(* PLC project flask_motion_app, Dassault Systèmes ControlBuild 2021x HF2 *)
(* stored: creationDateTime 2023-10-03T16:51:02-01:00 *)

CONFIGURATION flask_motion_app
  VAR_GLOBAL
    weight AT 523 : INT := 150;
    masterPosition AT 17 : REAL := 0.0;
    plc/presConvUp AT 6 : BOOL := false;
    plc/presConvDw AT 7 : BOOL := false;
    plc/masterPosition AT 17 : REAL := 0.0;
    plc/idRead AT 525 : INT := 0;
    plc/mesuredWeight AT 526 : INT := 0;
    plc/bpStart AT 8 : BOOL := false;
    plc/bpAuto AT 9 : BOOL := false;
    plc/bpManu AT 10 : BOOL := false;
    plc/bpEmergencyStop AT 11 : BOOL := false;
    plc/bpStop AT 12 : BOOL := false;
    plc/HomeCmd AT 13 : BOOL := false;
    plc/MoveVelCmd AT 14 : BOOL := false;
    plc/MoveAbsCmd AT 15 : BOOL := false;
    plc/MoveVel1ManualCmd AT 16 : BOOL := false;
    plc/MoveVel2ManualCmd AT 17 : BOOL := false;
    plc/MoveAbs1ManualCmd AT 18 : BOOL := false;
    plc/MoveAbs2ManualCmd AT 19 : BOOL := false;
    plc/StopCmd AT 20 : BOOL := false;
    plc/MovePosition AT 32 : REAL := 0.0;
    plc/MoveSpeed AT 33 : REAL := 100.0;
    plc/MoveAcceleration AT 34 : REAL := 100.0;
    plc/MoveDeceleration AT 35 : REAL := 100.0;
    plc/offsetAxToMa AT 36 : REAL := 0.0;
    plc/gripSyringes AT 21 : BOOL := false;
    plc/Auto AT 22 : BOOL := false;
    plc/Manu AT 23 : BOOL := false;
    plc/run AT 24 : BOOL := false;
    plc/forwardUp AT 25 : BOOL := false;
    plc/backwardUp AT 26 : BOOL := false;
    plc/forwardDw AT 27 : BOOL := false;
    plc/backwardDw AT 28 : BOOL := false;
    plc/ejectBadProd AT 29 : BOOL := false;
    plc/modemanagement/bpStart AT 8 : BOOL := false;
    plc/modemanagement/bpAuto AT 9 : BOOL := false;
    plc/modemanagement/bpManu AT 10 : BOOL := false;
    plc/modemanagement/bpEmergencyStop AT 11 : BOOL := false;
    plc/modemanagement/bpStop AT 12 : BOOL := false;
    plc/modemanagement/Auto AT 22 : BOOL := false;
    plc/modemanagement/Manu AT 23 : BOOL := false;
    plc/modemanagement/run AT 24 : BOOL := false;
    plc/motors/Auto AT 22 : BOOL := false;
    plc/motors/Manu AT 23 : BOOL := false;
    plc/motors/run AT 24 : BOOL := false;
    plc/motors/presConvUp AT 6 : BOOL := false;
    plc/motors/presConvDw AT 7 : BOOL := false;
    plc/motors/masterPosition AT 17 : REAL := 0.0;
    plc/motors/mesuredWeight AT 526 : INT := 0;
    plc/motors/phaseCode AT 527 : INT := 0;
    plc/motors/forwardUp AT 25 : BOOL := false;
    plc/motors/backwardUp AT 26 : BOOL := false;
    plc/motors/forwardDw AT 27 : BOOL := false;
    plc/motors/backwardDw AT 28 : BOOL := false;
    plc/motors/ejectBadProd AT 29 : BOOL := false;
    plc/motors/weihtOk AT 30 : BOOL := false;
    plc/motors/upperLimitOk AT 32 : BOOL := false;
    plc/motors/lowerLimitOk AT 33 : BOOL := false;
    plc/motors/prtSensorConvDw AT 529 : TIME := T#0h0m0s500ms;
    plc/motors/prtSensorConvUp AT 533 : TIME := T#0h0m1s500ms;
    plc/motors/upperLimitWeight AT 537 : INT := 125;
    plc/motors/lowerLimitWeight AT 538 : INT := 115;
    plc/robotctrl/forwardUp AT 25 : BOOL := false;
    plc/robotctrl/backwardUp AT 26 : BOOL := false;
    plc/robotctrl/forwardDw AT 27 : BOOL := false;
    plc/robotctrl/backwardDw AT 28 : BOOL := false;
    plc/robotctrl/presConvUp AT 6 : BOOL := false;
    plc/robotctrl/presConvDw AT 7 : BOOL := false;
    plc/robotctrl/masterPosition AT 17 : REAL := 0.0;
    plc/robotctrl/Auto AT 22 : BOOL := false;
    plc/robotctrl/Manu AT 23 : BOOL := false;
    plc/robotctrl/run AT 24 : BOOL := false;
    plc/robotctrl/weightOk AT 30 : BOOL := false;
    plc/robotctrl/phaseCode AT 527 : INT := 0;
    plc/robotctrl/HomeCmd AT 13 : BOOL := false;
    plc/robotctrl/MoveVelCmd AT 14 : BOOL := false;
    plc/robotctrl/MoveAbsCmd AT 15 : BOOL := false;
    plc/robotctrl/MoveVel1ManualCmd AT 16 : BOOL := false;
    plc/robotctrl/MoveVel2ManualCmd AT 17 : BOOL := false;
    plc/robotctrl/MoveAbs1ManualCmd AT 18 : BOOL := false;
    plc/robotctrl/MoveAbs2ManualCmd AT 19 : BOOL := false;
    plc/robotctrl/StopCmd AT 20 : BOOL := false;
    plc/robotctrl/MovePosition AT 32 : REAL := 0.0;
    plc/robotctrl/MoveSpeed AT 33 : REAL := 100.0;
    plc/robotctrl/MoveAcceleration AT 34 : REAL := 100.0;
    plc/robotctrl/MoveDeceleration AT 35 : REAL := 100.0;
    plc/robotctrl/offsetAxToMa AT 36 : REAL := 0.0;
    plc/robotctrl/gripSyringes AT 21 : BOOL := false;
    plc/robotctrl/endPhase1 AT 37 : REAL := 50.0;
    plc/robotctrl/endPhase2 AT 38 : REAL := 60.0;
    plc/robotctrl/endPhase3 AT 39 : REAL := 150.0;
    plc/robotctrl/endPhase4 AT 40 : REAL := 200.0;
    plc/robotctrl/speedPhase1 AT 41 : REAL := 80.0;
    plc/robotctrl/speedPhase2 AT 42 : REAL := 85.0;
    plc/robotctrl/speedPhase3 AT 43 : REAL := 100.0;
    plc/robotctrl/speedPhase4 AT 44 : REAL := 100.0;
    plc/robotctrl/globalSpeedFactor AT 45 : REAL := 100.0;
    robot6axis_ctrled1/armOrigin AT 27 : ARRAY[1..3] OF REAL := [800.0, 400.0, 0.0];
    robot6axis_ctrled1/profileNr AT 524 : DINT := 0;
    robot6axis_ctrled1/HomeCmd AT 13 : BOOL := false;
    robot6axis_ctrled1/MoveVelCmd AT 14 : BOOL := false;
    robot6axis_ctrled1/MoveAbsCmd AT 15 : BOOL := false;
    robot6axis_ctrled1/MoveVel1ManualCmd AT 16 : BOOL := false;
    robot6axis_ctrled1/MoveVel2ManualCmd AT 17 : BOOL := false;
    robot6axis_ctrled1/MoveAbs1ManualCmd AT 18 : BOOL := false;
    robot6axis_ctrled1/MoveAbs2ManualCmd AT 19 : BOOL := false;
    robot6axis_ctrled1/StopCmd AT 20 : BOOL := false;
    robot6axis_ctrled1/MovePosition AT 32 : REAL := 0.0;
    robot6axis_ctrled1/MoveSpeed AT 33 : REAL := 100.0;
    robot6axis_ctrled1/MoveAcceleration AT 34 : REAL := 100.0;
    robot6axis_ctrled1/MoveDeceleration AT 35 : REAL := 100.0;
    robot6axis_ctrled1/offsetAxToMa AT 36 : REAL := 0.0;
    robot6axis_ctrled1/gripSyringes AT 21 : BOOL := false;
    robot6axis_ctrled1/Auto AT 22 : BOOL := false;
    robot6axis_ctrled1/Manu AT 23 : BOOL := false;
    robot6axis_ctrled1/run AT 24 : BOOL := false;
    robot6axis_ctrled1/armExtrem AT 22 : ARRAY[1..3] OF REAL := [3(0.0)];
    robot6axis_ctrled1/velX AT 21 : REAL := 0.0;
    robot6axis_ctrled1/velY AT 20 : REAL := 0.0;
    robot6axis_ctrled1/velZ AT 19 : REAL := 0.0;
    robot6axis_ctrled1/armInStop AT 5 : BOOL := false;
    robot6axis_ctrled1/masterPosition AT 17 : REAL := 0.0;
    robot6axis_ctrled1/ActualPositionAx AT 18 : REAL := 0.0;
    robot6axis_ctrled1/robot6axis_cams/profileNr AT 524 : DINT := 0;
    robot6axis_ctrled1/robot6axis_cams/HomeCmd AT 13 : BOOL := false;
    robot6axis_ctrled1/robot6axis_cams/MoveVelCmd AT 14 : BOOL := false;
    robot6axis_ctrled1/robot6axis_cams/MoveAbsCmd AT 15 : BOOL := false;
    robot6axis_ctrled1/robot6axis_cams/MoveVel1ManualCmd AT 16 : BOOL := false;
    robot6axis_ctrled1/robot6axis_cams/MoveVel2ManualCmd AT 17 : BOOL := false;
    robot6axis_ctrled1/robot6axis_cams/MoveAbs1ManualCmd AT 18 : BOOL := false;
    robot6axis_ctrled1/robot6axis_cams/MoveAbs2ManualCmd AT 19 : BOOL := false;
    robot6axis_ctrled1/robot6axis_cams/StopCmd AT 20 : BOOL := false;
    robot6axis_ctrled1/robot6axis_cams/MovePosition AT 32 : REAL := 0.0;
    robot6axis_ctrled1/robot6axis_cams/MoveSpeed AT 33 : REAL := 100.0;
    robot6axis_ctrled1/robot6axis_cams/MoveAcceleration AT 34 : REAL := 100.0;
    robot6axis_ctrled1/robot6axis_cams/MoveDeceleration AT 35 : REAL := 100.0;
    robot6axis_ctrled1/robot6axis_cams/offsetAxToMa AT 36 : REAL := 0.0;
    robot6axis_ctrled1/robot6axis_cams/name1 AT 636 : STRING(50) := 'CamAxis1_exa.txt';
    robot6axis_ctrled1/robot6axis_cams/name2 AT 583 : STRING(50) := 'CamAxis2_exa.txt';
    robot6axis_ctrled1/robot6axis_cams/name3 AT 530 : STRING(50) := 'CamAxis3_exa.txt';
    robot6axis_ctrled1/robot6axis_cams/name4 AT 477 : STRING(50) := 'CamAxis4_exa.txt';
    robot6axis_ctrled1/robot6axis_cams/name5 AT 424 : STRING(50) := 'CamAxis5_exa.txt';
    robot6axis_ctrled1/robot6axis_cams/name6 AT 371 : STRING(50) := 'CamAxis6_exa.txt';
    robot6axis_ctrled1/robot6axis_cams/name1_rej AT 318 : STRING(50) := 'CamAxis1_rej.txt';
    robot6axis_ctrled1/robot6axis_cams/name2_rej AT 265 : STRING(50) := 'CamAxis2_rej.txt';
    robot6axis_ctrled1/robot6axis_cams/name3_rej AT 212 : STRING(50) := 'CamAxis3_rej.txt';
    robot6axis_ctrled1/robot6axis_cams/name4_rej AT 159 : STRING(50) := 'CamAxis4_rej.txt';
    robot6axis_ctrled1/robot6axis_cams/name5_rej AT 106 : STRING(50) := 'CamAxis5_rej.txt';
    robot6axis_ctrled1/robot6axis_cams/name6_rej AT 53 : STRING(50) := 'CamAxis6_rej.txt';
    robot6axis_ctrled1/robot6axis_cams/slavePosition1 AT 167 : REAL := 0.0;
    robot6axis_ctrled1/robot6axis_cams/slavePosition2 AT 168 : REAL := 0.0;
    robot6axis_ctrled1/robot6axis_cams/slavePosition3 AT 169 : REAL := 0.0;
    robot6axis_ctrled1/robot6axis_cams/slavePosition4 AT 170 : REAL := 0.0;
    robot6axis_ctrled1/robot6axis_cams/slavePosition5 AT 171 : REAL := 0.0;
    robot6axis_ctrled1/robot6axis_cams/slavePosition6 AT 172 : REAL := 0.0;
    robot6axis_ctrled1/robot6axis_cams/ActualPositionAx AT 18 : REAL := 0.0;
    robot6axis_ctrled1/robot6axis_cams/masterPosition AT 17 : REAL := 0.0;
    robot6axis_ctrled1/robot6axis_cams/servo_kinetix2/status AT 583 : INT := 0;
    robot6axis_ctrled1/robot6axis_cams/servo_kinetix2/errorFlag AT 582 : INT := 0;
    robot6axis_ctrled1/robot6axis_cams/servo_kinetix2/ActualPositionAx1 AT 2639 : REAL := 0.0;
    robot6axis_ctrled1/robot6axis_cams/servo_kinetix2/MoveVelDone1 AT 108 : BOOL := false;
    robot6axis_ctrled1/robot6axis_cams/servo_kinetix2/ActualVelocity1 AT 2638 : REAL := 0.0;
    robot6axis_ctrled1/robot6axis_cams/servo_kinetix2/MoveAbsDone1 AT 107 : BOOL := false;
    robot6axis_ctrled1/robot6axis_cams/servo_kinetix2/HomeCmd AT 13 : BOOL := false;
    robot6axis_ctrled1/robot6axis_cams/servo_kinetix2/MoveVelCmd AT 14 : BOOL := false;
    robot6axis_ctrled1/robot6axis_cams/servo_kinetix2/MoveAbsCmd AT 15 : BOOL := false;
    robot6axis_ctrled1/robot6axis_cams/servo_kinetix2/MoveVel1ManualCmd AT 16 : BOOL := false;
    robot6axis_ctrled1/robot6axis_cams/servo_kinetix2/MoveVel2ManualCmd AT 17 : BOOL := false;
    robot6axis_ctrled1/robot6axis_cams/servo_kinetix2/MoveAbs1ManualCmd AT 18 : BOOL := false;
    robot6axis_ctrled1/robot6axis_cams/servo_kinetix2/MoveAbs2ManualCmd AT 19 : BOOL := false;
    robot6axis_ctrled1/robot6axis_cams/servo_kinetix2/StopCmd AT 20 : BOOL := false;
    robot6axis_ctrled1/robot6axis_cams/servo_kinetix2/MovePosition AT 32 : REAL := 0.0;
    robot6axis_ctrled1/robot6axis_cams/servo_kinetix2/MoveSpeed AT 33 : REAL := 100.0;
    robot6axis_ctrled1/robot6axis_cams/servo_kinetix2/MoveAcceleration AT 34 : REAL := 100.0;
    robot6axis_ctrled1/robot6axis_cams/servo_kinetix2/MoveDeceleration AT 35 : REAL := 100.0;
    robot6axis_ctrled1/robot6axis_cams/servo_kinetix2/offsetAxToMa AT 36 : REAL := 0.0;
    robot6axis_ctrled1/robot6axis_cams/servo_kinetix2/PLC_StatusReady AT 106 : BOOL := true;
    robot6axis_ctrled1/robot6axis_cams/servo_kinetix2/PLC_StatusMoved AT 105 : BOOL := false;
    robot6axis_ctrled1/robot6axis_cams/servo_kinetix2/PLC_StatusStand AT 104 : BOOL := false;
    robot6axis_ctrled1/robot6axis_cams/servo_kinetix2/PLC_ActualPositionAx AT 2637 : REAL := 0.0;
    robot6axis_ctrled1/robot6axis_cams/servo_kinetix2/PLC_ActualPositionMa AT 2636 : REAL := 0.0;
    robot6axis_ctrled1/robot6axis_cams/servo_kinetix2/PLC_ActualVelocity AT 2635 : REAL := 0.0;
    robot6axis_ctrled1/robot6axis_cams/servo_kinetix2/physicalPosInit AT 2634 : REAL := 0.0;
    robot6axis_ctrled1/robot6axis_cams/servo_kinetix2/MAX_SPEED AT 2633 : REAL(0.0..3.4e+038) := 50.0;
    robot6axis_ctrled1/robot6axis_cams/servo_kinetix2/MAX_ACCEL AT 2632 : REAL(0.0..3.4e+038) := 1500.0;
    robot6axis_ctrled1/robot6axis_cams/servo_kinetix2/MAX_DECEL AT 2631 : REAL(0.0..3.4e+038) := 1500.0;
    robot6axis_ctrled1/robot6axis_cams/servo_kinetix2/MODULO_LENGTH AT 2630 : REAL := 0.0;
    robot6axis_ctrled1/robot6axis_cams/servo_kinetix2/StatusReady AT 103 : BOOL := true;
    robot6axis_ctrled1/robot6axis_cams/servo_kinetix2/StatusMoved AT 102 : BOOL := false;
    robot6axis_ctrled1/robot6axis_cams/servo_kinetix2/StatusStand AT 101 : BOOL := false;
    robot6axis_ctrled1/robot6axis_cams/servo_kinetix2/ActualPositionAx AT 18 : REAL := 0.0;
    robot6axis_ctrled1/robot6axis_cams/servo_kinetix2/ActualPositionMa AT 2629 : REAL := 0.0;
    robot6axis_ctrled1/robot6axis_cams/servo_kinetix2/ActualVelocity AT 2628 : REAL := 0.0;
    robot6axis_ctrled1/robot6axis_cams/servo_kinetix2/MaximumVelocity AT 2627 : REAL := 0.0;
    robot6axis_ctrled1/robot6axis_cams/servo_kinetix2/StatusPosIncrease AT 100 : BOOL := false;
    robot6axis_ctrled1/robot6axis_cams/servo_kinetix2/StatusPosDecrease AT 99 : BOOL := false;
    robot6axis_ctrled1/robot6axis_cams/servo_kinetix2/displayJauge AT 2626 : REAL := 0.0;
    robot6axis_ctrled1/robot6axis_cams/servo_kinetix2/servo_mode/PLC_StatusReady AT 106 : BOOL := true;
    robot6axis_ctrled1/robot6axis_cams/servo_kinetix2/servo_mode/PLC_StatusMoved AT 105 : BOOL := false;
    robot6axis_ctrled1/robot6axis_cams/servo_kinetix2/servo_mode/PLC_StatusStand AT 104 : BOOL := false;
    robot6axis_ctrled1/robot6axis_cams/servo_kinetix2/servo_mode/PLC_ActualPositionAx AT 2637 : REAL := 0.0;
    robot6axis_ctrled1/robot6axis_cams/servo_kinetix2/servo_mode/PLC_ActualPositionMa AT 2636 : REAL := 0.0;
    robot6axis_ctrled1/robot6axis_cams/servo_kinetix2/servo_mode/PLC_ActualVelocity AT 2635 : REAL := 0.0;
    robot6axis_ctrled1/robot6axis_cams/servo_kinetix2/servo_mode/StatusReady AT 109 : BOOL := true;
    robot6axis_ctrled1/robot6axis_cams/servo_kinetix2/servo_mode/StatusMoved AT 110 : BOOL := false;
    robot6axis_ctrled1/robot6axis_cams/servo_kinetix2/servo_mode/StatusStand AT 111 : BOOL := false;
    robot6axis_ctrled1/robot6axis_cams/servo_kinetix2/servo_mode/ActualPositionMa AT 5088 : REAL := 0.0;
    robot6axis_ctrled1/robot6axis_cams/servo_kinetix2/servo_mode/ActualVelocity AT 5089 : REAL := 0.0;
    robot6axis_ctrled1/robot6axis_cams/servo_kinetix2/servo_mode/MaximumVelocity AT 5090 : REAL := 0.0;
    robot6axis_ctrled1/robot6axis_cams/servo_kinetix2/servo_mode/physicalPosInit AT 2634 : REAL := 0.0;
    robot6axis_ctrled1/robot6axis_cams/servo_kinetix2/servo_mode/ActualPositionAx AT 2639 : REAL := 0.0;
    robot6axis_ctrled1/robot6axis_cams/servo_kinetix2/servo_mode/StatusReady_o AT 103 : BOOL := true;
    robot6axis_ctrled1/robot6axis_cams/servo_kinetix2/servo_mode/StatusMoved_o AT 102 : BOOL := false;
    robot6axis_ctrled1/robot6axis_cams/servo_kinetix2/servo_mode/StatusStand_o AT 101 : BOOL := false;
    robot6axis_ctrled1/robot6axis_cams/servo_kinetix2/servo_mode/ActualPositionAx_o AT 18 : REAL := 0.0;
    robot6axis_ctrled1/robot6axis_cams/servo_kinetix2/servo_mode/ActualPositionMa_o AT 2629 : REAL := 0.0;
    robot6axis_ctrled1/robot6axis_cams/servo_kinetix2/servo_mode/ActualVelocity_o AT 2628 : REAL := 0.0;
    robot6axis_ctrled1/robot6axis_cams/servo_kinetix2/servo_mode/MaximumVelocity_o AT 2627 : REAL := 0.0;
    robot6axis_ctrled1/robot6axis_cams/servo_kinetix2/servo_mode/StatusPosIncrease_o AT 100 : BOOL := false;
    robot6axis_ctrled1/robot6axis_cams/servo_kinetix2/servo_mode/StatusPosDecrease_o AT 99 : BOOL := false;
    robot6axis_ctrled1/robot6axis_cams/servo_kinetix2/servo_mode/displayJauge_o AT 2626 : REAL := 0.0;
    robot6axis_ctrled1/robot6axis_cams/servo_kinetix2/servo_mode/PLCMode AT 116 : BOOL := false;
    robot6axis_ctrled1/robot6axis_cams/servo_kinetix2/servo_mode/PLCMode1 AT 117 : BOOL := false;
    robot6axis_ctrled1/robot6axis_cams/servo_kinetix2/servo_mode/initDone AT 118 : BOOL := false;
    robot6axis_ctrled1/robot6axis_cams/servo_kinetix2/servo_mode/displayPosMin AT 5093 : REAL := 0.0;
    robot6axis_ctrled1/robot6axis_cams/servo_kinetix2/servo_mode/displayPosMax AT 5094 : REAL := 0.0;
    robot6axis_ctrled1/robot6axis_cams/servo_kinetix2/servo_mode/PLC_ActualPositionAx1 AT 5095 : REAL := 0.0;
    robot6axis_ctrled1/robot6axis_cams/servo_kinetix2/servo_mode/PLC_ActualVelocity1 AT 5096 : REAL := 0.0;
    robot6axis_ctrled1/robot6axis_cams/servo_kinetix2/servo_mode/ActualPositionAx1 AT 5097 : REAL := 0.0;
    robot6axis_ctrled1/robot6axis_cams/servo_kinetix2/servo_mode/ActualVelocity1 AT 5098 : REAL := 0.0;
    robot6axis_ctrled1/robot6axis_cams/servo_kinetix2/servo_mode/offsetAxToMa AT 5099 : REAL := 0.0;
    robot6axis_ctrled1/robot6axis_cams/servo_kinetix2/servo_mode/offsetAxToMa1 AT 5100 : REAL := 0.0;
    robot6axis_ctrled1/robot6axis_cams/servo_kinetix2/servo_mode/ActualPositionMa_o1 AT 5101 : REAL := 0.0;
    robot6axis_ctrled1/robot6axis_cams/servo_kinetix2/servo_control/HomeCmd AT 13 : BOOL := false;
    robot6axis_ctrled1/robot6axis_cams/servo_kinetix2/servo_control/MoveVelCmd AT 14 : BOOL := false;
    robot6axis_ctrled1/robot6axis_cams/servo_kinetix2/servo_control/MoveAbsCmd AT 15 : BOOL := false;
    robot6axis_ctrled1/robot6axis_cams/servo_kinetix2/servo_control/MoveVel1ManualCmd AT 16 : BOOL := false;
    robot6axis_ctrled1/robot6axis_cams/servo_kinetix2/servo_control/MoveVel2ManualCmd AT 17 : BOOL := false;
    robot6axis_ctrled1/robot6axis_cams/servo_kinetix2/servo_control/MoveAbs1ManualCmd AT 18 : BOOL := false;
    robot6axis_ctrled1/robot6axis_cams/servo_kinetix2/servo_control/MoveAbs2ManualCmd AT 19 : BOOL := false;
    robot6axis_ctrled1/robot6axis_cams/servo_kinetix2/servo_control/StopCmd AT 20 : BOOL := false;
    robot6axis_ctrled1/robot6axis_cams/servo_kinetix2/servo_control/MovePosition AT 32 : REAL := 0.0;
    robot6axis_ctrled1/robot6axis_cams/servo_kinetix2/servo_control/MoveSpeed AT 33 : REAL := 100.0;
    robot6axis_ctrled1/robot6axis_cams/servo_kinetix2/servo_control/MoveAcceleration AT 34 : REAL := 100.0;
    robot6axis_ctrled1/robot6axis_cams/servo_kinetix2/servo_control/MoveDeceleration AT 35 : REAL := 100.0;
    robot6axis_ctrled1/robot6axis_cams/servo_kinetix2/servo_control/offsetAxToMa AT 36 : REAL := 0.0;
    robot6axis_ctrled1/robot6axis_cams/servo_kinetix2/servo_control/physicalPosInit AT 2634 : REAL := 0.0;
    robot6axis_ctrled1/robot6axis_cams/servo_kinetix2/servo_control/MAX_SPEED AT 2633 : REAL(0.0..3.4e+038) := 50.0;
    robot6axis_ctrled1/robot6axis_cams/servo_kinetix2/servo_control/status AT 583 : INT := 0;
    robot6axis_ctrled1/robot6axis_cams/servo_kinetix2/servo_control/errorFlag AT 582 : INT := 0;
    robot6axis_ctrled1/robot6axis_cams/servo_kinetix2/servo_control/IOActualPositionAx AT 2639 : REAL := 0.0;
    robot6axis_ctrled1/robot6axis_cams/servo_kinetix2/servo_control/IOVelDone AT 108 : BOOL := false;
    robot6axis_ctrled1/robot6axis_cams/servo_kinetix2/servo_control/IOAbsDone AT 107 : BOOL := false;
    robot6axis_ctrled1/robot6axis_cams/servo_kinetix2/servo_control/IOActualVelocity AT 2638 : REAL := 0.0;
    robot6axis_ctrled1/robot6axis_cams/servo_kinetix2/servo_control/OperationMode AT 608 : INT := 0;
    robot6axis_ctrled1/robot6axis_cams/servo_kinetix2/servo_control/StatusReady AT 109 : BOOL := true;
    robot6axis_ctrled1/robot6axis_cams/servo_kinetix2/servo_control/StatusMove AT 110 : BOOL := false;
    robot6axis_ctrled1/robot6axis_cams/servo_kinetix2/servo_control/StatusStand AT 111 : BOOL := false;
    robot6axis_ctrled1/robot6axis_cams/servo_kinetix2/servo_control/ActualPositionMa AT 5088 : REAL := 0.0;
    robot6axis_ctrled1/robot6axis_cams/servo_kinetix2/servo_control/ActualVelocity AT 5089 : REAL := 0.0;
    robot6axis_ctrled1/robot6axis_cams/servo_kinetix2/servo_control/MaximumVelocity AT 5090 : REAL := 0.0;
    robot6axis_ctrled1/robot6axis_cams/servo_kinetix2/servo_control/VelEnabled AT 112 : BOOL := false;
    robot6axis_ctrled1/robot6axis_cams/servo_kinetix2/servo_control/VelCmd AT 113 : BOOL := false;
    robot6axis_ctrled1/robot6axis_cams/servo_kinetix2/servo_control/PosEnabled AT 114 : BOOL := false;
    robot6axis_ctrled1/robot6axis_cams/servo_kinetix2/servo_control/PosCmd AT 115 : BOOL := false;
    robot6axis_ctrled1/robot6axis_cams/servo_kinetix2/servo_control/Position AT 5092 : REAL := 0.0;
    robot6axis_ctrled1/robot6axis_cams/servo_kinetix2/servo_control/Speed AT 5091 : REAL := 0.0;
    robot6axis_ctrled1/robot6axis_cams/servo_kinetix2/servo_control/ManualMode AT 609 : INT := 0;
    robot6axis_ctrled1/robot6axis_cams/servo_kinetix2/servo_control/initDone AT 119 : BOOL := false;
    robot6axis_ctrled1/robot6axis_cams/servo_kinetix2/servo_control/ActualPositionMa1 AT 5102 : REAL := 0.0;
    robot6axis_ctrled1/robot6axis_cams/servo_kinetix2/servo_control/offsetAxToMa1 AT 5103 : REAL := 0.0;
    robot6axis_ctrled1/robot6axis_cams/servo_kinetix2/servo_control/HOME_POSITION AT 5104 : REAL := 100.0;
    robot6axis_ctrled1/robot6axis_cams/servo_kinetix2/servo_control/MANUAL_POSITION1 AT 5105 : REAL := 0.0;
    robot6axis_ctrled1/robot6axis_cams/servo_kinetix2/servo_control/MANUAL_POSITION2 AT 5106 : REAL := 150.0;
    robot6axis_ctrled1/robot6axis_cams/servo_kinetix2/servo_control/MANUAL_SPEED1 AT 5107 : REAL := -100.0;
    robot6axis_ctrled1/robot6axis_cams/servo_kinetix2/servo_control/MANUAL_SPEED2 AT 5108 : REAL := 100.0;
    robot6axis_ctrled1/robot6axis_cams/servo_kinetix2/servo_control/MANUAL_SPEED AT 5109 : REAL := 100.0;
    robot6axis_ctrled1/robot6axis_cams/servo_kinetix2/servo_velocity/MoveVelEnable AT 112 : BOOL := false;
    robot6axis_ctrled1/robot6axis_cams/servo_kinetix2/servo_velocity/MoveVelStart AT 113 : BOOL := false;
    robot6axis_ctrled1/robot6axis_cams/servo_kinetix2/servo_velocity/MoveSpeed AT 5091 : REAL := 0.0;
    robot6axis_ctrled1/robot6axis_cams/servo_kinetix2/servo_velocity/MoveAcceleration AT 34 : REAL := 100.0;
    robot6axis_ctrled1/robot6axis_cams/servo_kinetix2/servo_velocity/MoveDeceleration AT 35 : REAL := 100.0;
    robot6axis_ctrled1/robot6axis_cams/servo_kinetix2/servo_velocity/MAX_SPEED AT 2633 : REAL(0.0..3.4e+038) := 50.0;
    robot6axis_ctrled1/robot6axis_cams/servo_kinetix2/servo_velocity/MAX_ACCEL AT 2632 : REAL(0.0..3.4e+038) := 1500.0;
    robot6axis_ctrled1/robot6axis_cams/servo_kinetix2/servo_velocity/MAX_DECEL AT 2631 : REAL(0.0..3.4e+038) := 1500.0;
    robot6axis_ctrled1/robot6axis_cams/servo_kinetix2/servo_velocity/MODULO_LENGTH AT 2630 : REAL := 0.0;
    robot6axis_ctrled1/robot6axis_cams/servo_kinetix2/servo_velocity/status AT 583 : INT := 0;
    robot6axis_ctrled1/robot6axis_cams/servo_kinetix2/servo_velocity/errorFlag AT 582 : INT := 0;
    robot6axis_ctrled1/robot6axis_cams/servo_kinetix2/servo_velocity/MoveVelDone AT 108 : BOOL := false;
    robot6axis_ctrled1/robot6axis_cams/servo_kinetix2/servo_velocity/ActualPositionAx AT 2639 : REAL := 0.0;
    robot6axis_ctrled1/robot6axis_cams/servo_kinetix2/servo_velocity/ActualVelocity AT 2638 : REAL := 0.0;
    robot6axis_ctrled1/robot6axis_cams/servo_kinetix2/servo_velocity/firstStep AT 120 : BOOL := true;
    robot6axis_ctrled1/robot6axis_cams/servo_kinetix2/servo_velocity/stepDone AT 121 : BOOL := false;
    robot6axis_ctrled1/robot6axis_cams/servo_kinetix2/servo_velocity/currentTime AT 5110 : REAL := 0.0;
    robot6axis_ctrled1/robot6axis_cams/servo_kinetix2/servo_velocity/MoveSpeed1 AT 5111 : REAL := 0.0;
    robot6axis_ctrled1/robot6axis_cams/servo_kinetix2/servo_velocity/acceleration AT 5112 : REAL := 0.0;
    robot6axis_ctrled1/robot6axis_cams/servo_kinetix2/servo_velocity/deceleration AT 5113 : REAL := 0.0;
    robot6axis_ctrled1/robot6axis_cams/servo_kinetix2/servo_velocity/orderSpeed AT 5114 : REAL := 0.0;
    robot6axis_ctrled1/robot6axis_cams/servo_kinetix2/servo_velocity/endChangeSpeed AT 5115 : REAL := 0.0;
    robot6axis_ctrled1/robot6axis_cams/servo_kinetix2/servo_velocity/accelDecelChangeSpeed AT 5116 : REAL := 0.0;
    robot6axis_ctrled1/robot6axis_cams/servo_kinetix2/servo_velocity/ActualVelocity1 AT 5117 : REAL := 0.0;
    robot6axis_ctrled1/robot6axis_cams/servo_kinetix2/servo_velocity/speedChanged AT 122 : BOOL := false;
    robot6axis_ctrled1/robot6axis_cams/servo_kinetix2/servo_position/MoveAbsEnable AT 114 : BOOL := false;
    robot6axis_ctrled1/robot6axis_cams/servo_kinetix2/servo_position/MoveAbsStart AT 115 : BOOL := false;
    robot6axis_ctrled1/robot6axis_cams/servo_kinetix2/servo_position/MovePosition AT 5092 : REAL := 0.0;
    robot6axis_ctrled1/robot6axis_cams/servo_kinetix2/servo_position/MoveSpeed AT 5091 : REAL := 0.0;
    robot6axis_ctrled1/robot6axis_cams/servo_kinetix2/servo_position/MoveAcceleration AT 34 : REAL := 100.0;
    robot6axis_ctrled1/robot6axis_cams/servo_kinetix2/servo_position/MoveDeceleration AT 35 : REAL := 100.0;
    robot6axis_ctrled1/robot6axis_cams/servo_kinetix2/servo_position/MAX_SPEED AT 2633 : REAL(0.0..3.4e+038) := 50.0;
    robot6axis_ctrled1/robot6axis_cams/servo_kinetix2/servo_position/MAX_ACCEL AT 2632 : REAL(0.0..3.4e+038) := 1500.0;
    robot6axis_ctrled1/robot6axis_cams/servo_kinetix2/servo_position/MAX_DECEL AT 2631 : REAL(0.0..3.4e+038) := 1500.0;
    robot6axis_ctrled1/robot6axis_cams/servo_kinetix2/servo_position/MODULO_LENGTH AT 2630 : REAL := 0.0;
    robot6axis_ctrled1/robot6axis_cams/servo_kinetix2/servo_position/status AT 583 : INT := 0;
    robot6axis_ctrled1/robot6axis_cams/servo_kinetix2/servo_position/errorFlag AT 582 : INT := 0;
    robot6axis_ctrled1/robot6axis_cams/servo_kinetix2/servo_position/MoveAbsDone AT 107 : BOOL := false;
    robot6axis_ctrled1/robot6axis_cams/servo_kinetix2/servo_position/ActualPositionAx AT 2639 : REAL := 0.0;
    robot6axis_ctrled1/robot6axis_cams/servo_kinetix2/servo_position/ActualVelocity AT 2638 : REAL := 0.0;
    robot6axis_ctrled1/robot6axis_cams/servo_kinetix2/servo_position/firstStep AT 123 : BOOL := true;
    robot6axis_ctrled1/robot6axis_cams/servo_kinetix2/servo_position/stepDone AT 124 : BOOL := false;
    robot6axis_ctrled1/robot6axis_cams/servo_kinetix2/servo_position/timeToStop AT 5118 : REAL := 0.0;
    robot6axis_ctrled1/robot6axis_cams/servo_kinetix2/servo_position/distanceToStop AT 5119 : REAL := 0.0;
    robot6axis_ctrled1/robot6axis_cams/servo_kinetix2/servo_position/distance AT 5120 : REAL := 0.0;
    robot6axis_ctrled1/robot6axis_cams/servo_kinetix2/servo_position/currentTime AT 5121 : REAL := 0.0;
    robot6axis_ctrled1/robot6axis_cams/servo_kinetix2/servo_position/currentSpeed1 AT 5122 : REAL := 0.0;
    robot6axis_ctrled1/robot6axis_cams/servo_kinetix2/servo_position/targetPosition AT 5123 : REAL := 0.0;
    robot6axis_ctrled1/robot6axis_cams/servo_kinetix2/servo_position/ActualPositionAx1 AT 5124 : REAL := 0.0;
    robot6axis_ctrled1/robot6axis_cams/servo_kinetix2/servo_position/acceleration AT 5125 : REAL := 0.0;
    robot6axis_ctrled1/robot6axis_cams/servo_kinetix2/servo_position/deceleration AT 5126 : REAL := 0.0;
    robot6axis_ctrled1/robot6axis_cams/servo_kinetix2/servo_position/orderSpeed AT 5127 : REAL := 0.0;
    robot6axis_ctrled1/robot6axis_cams/servo_kinetix2/servo_position/moveDirection AT 5128 : REAL := 0.0;
    robot6axis_ctrled1/robot6axis_cams/servo_kinetix2/servo_position/moveDirection1 AT 5129 : REAL := 0.0;
    robot6axis_ctrled1/robot6axis_cams/servo_kinetix2/servo_position/endChangeSpeed AT 5130 : REAL := 0.0;
    robot6axis_ctrled1/robot6axis_cams/servo_kinetix2/servo_position/ActualVelocity1 AT 5131 : REAL := 0.0;
    robot6axis_ctrled1/robot6axis_cams/cam_profile1/name AT 636 : STRING(50) := 'CamAxis1_exa.txt';
    robot6axis_ctrled1/robot6axis_cams/cam_profile1/nbPoints AT 584 : INT := 0;
    robot6axis_ctrled1/robot6axis_cams/cam_profile1/MasterPoints AT 2640 : ARRAY[1..100] OF REAL := [100(0.0)];
    robot6axis_ctrled1/robot6axis_cams/cam_profile1/SlavePoints AT 2742 : ARRAY[1..100] OF REAL := [100(0.0)];
    robot6axis_ctrled1/robot6axis_cams/cam_profile1/pointer AT 585 : DINT := 0;
    robot6axis_ctrled1/robot6axis_cams/cam_profile1/initialized AT 125 : BOOL := false;
    robot6axis_ctrled1/robot6axis_cams/cam_profile1/pFile AT 610 : DINT := 0;
    robot6axis_ctrled1/robot6axis_cams/cam_profile1/fault_reading AT 126 : BOOL := false;
    robot6axis_ctrled1/robot6axis_cams/cam_profile1/fault_openning AT 127 : BOOL := false;
    robot6axis_ctrled1/robot6axis_cams/cam_profile1/complete_path AT 689 : STRING(254) := '';
    robot6axis_ctrled1/robot6axis_cams/cam_profile7/name AT 318 : STRING(50) := 'CamAxis1_rej.txt';
    robot6axis_ctrled1/robot6axis_cams/cam_profile7/nbPoints AT 586 : INT := 0;
    robot6axis_ctrled1/robot6axis_cams/cam_profile7/MasterPoints AT 2844 : ARRAY[1..100] OF REAL := [100(0.0)];
    robot6axis_ctrled1/robot6axis_cams/cam_profile7/SlavePoints AT 2946 : ARRAY[1..100] OF REAL := [100(0.0)];
    robot6axis_ctrled1/robot6axis_cams/cam_profile7/pointer AT 587 : DINT := 0;
    robot6axis_ctrled1/robot6axis_cams/cam_profile7/initialized AT 128 : BOOL := false;
    robot6axis_ctrled1/robot6axis_cams/cam_profile7/pFile AT 611 : DINT := 0;
    robot6axis_ctrled1/robot6axis_cams/cam_profile7/fault_reading AT 129 : BOOL := false;
    robot6axis_ctrled1/robot6axis_cams/cam_profile7/fault_openning AT 130 : BOOL := false;
    robot6axis_ctrled1/robot6axis_cams/cam_profile7/complete_path AT 946 : STRING(254) := '';
    robot6axis_ctrled1/robot6axis_cams/cam_computation1/profileNr AT 524 : DINT := 0;
    robot6axis_ctrled1/robot6axis_cams/cam_computation1/MasterPositionIn AT 18 : REAL := 0.0;
    robot6axis_ctrled1/robot6axis_cams/cam_computation1/nbPoints0 AT 584 : INT := 0;
    robot6axis_ctrled1/robot6axis_cams/cam_computation1/MasterPoints0 AT 2640 : ARRAY[1..100] OF REAL := [100(0.0)];
    robot6axis_ctrled1/robot6axis_cams/cam_computation1/SlavePoints0 AT 2742 : ARRAY[1..100] OF REAL := [100(0.0)];
    robot6axis_ctrled1/robot6axis_cams/cam_computation1/pointer0 AT 585 : DINT := 0;
    robot6axis_ctrled1/robot6axis_cams/cam_computation1/nbPoints1 AT 586 : INT := 0;
    robot6axis_ctrled1/robot6axis_cams/cam_computation1/MasterPoints1 AT 2844 : ARRAY[1..100] OF REAL := [100(0.0)];
    robot6axis_ctrled1/robot6axis_cams/cam_computation1/SlavePoints1 AT 2946 : ARRAY[1..100] OF REAL := [100(0.0)];
    robot6axis_ctrled1/robot6axis_cams/cam_computation1/pointer1 AT 587 : DINT := 0;
    robot6axis_ctrled1/robot6axis_cams/cam_computation1/nbPoints2 AT 581 : INT := 0;
    robot6axis_ctrled1/robot6axis_cams/cam_computation1/MasterPoints2 AT 2524 : ARRAY[1..100] OF REAL := [100(0.0)];
    robot6axis_ctrled1/robot6axis_cams/cam_computation1/SlavePoints2 AT 2422 : ARRAY[1..100] OF REAL := [100(0.0)];
    robot6axis_ctrled1/robot6axis_cams/cam_computation1/pointer2 AT 580 : DINT := 0;
    robot6axis_ctrled1/robot6axis_cams/cam_computation1/nbPoints3 AT 579 : INT := 0;
    robot6axis_ctrled1/robot6axis_cams/cam_computation1/MasterPoints3 AT 2320 : ARRAY[1..100] OF REAL := [100(0.0)];
    robot6axis_ctrled1/robot6axis_cams/cam_computation1/SlavePoints3 AT 2218 : ARRAY[1..100] OF REAL := [100(0.0)];
    robot6axis_ctrled1/robot6axis_cams/cam_computation1/pointer3 AT 578 : DINT := 0;
    robot6axis_ctrled1/robot6axis_cams/cam_computation1/slavePosition AT 167 : REAL := 0.0;
    robot6axis_ctrled1/robot6axis_cams/cam_computation1/masterPosition AT 17 : REAL := 0.0;
    robot6axis_ctrled1/robot6axis_cams/cam_computation1/i AT 612 : INT := 0;
    robot6axis_ctrled1/robot6axis_cams/cam_computation1/modulo AT 5132 : REAL := 0.0;
    robot6axis_ctrled1/robot6axis_cams/cam_computation1/divider AT 613 : INT := 0;
    robot6axis_ctrled1/robot6axis_cams/cam_computation1/faultProfileNr AT 131 : BOOL := false;
    robot6axis_ctrled1/robot6axis_cams/cam_computation1/faultMasterPositionOOB AT 132 : BOOL := false;
    robot6axis_ctrled1/robot6axis_cams/cam_computation1/faultLinComputation AT 133 : BOOL := false;
    robot6axis_ctrled1/robot6axis_cams/cam_computation1/nbPoints AT 614 : INT := 0;
    robot6axis_ctrled1/robot6axis_cams/cam_computation1/MasterPoints AT 5133 : ARRAY[1..100] OF REAL := [100(0.0)];
    robot6axis_ctrled1/robot6axis_cams/cam_computation1/SlavePoints AT 5235 : ARRAY[1..100] OF REAL := [100(0.0)];
    robot6axis_ctrled1/robot6axis_cams/cam_computation1/found AT 134 : BOOL := false;
    robot6axis_ctrled1/robot6axis_cams/cam_computation1/index AT 615 : INT := 0;
    robot6axis_ctrled1/robot6axis_cams/cam_computation1/linDenom AT 5337 : REAL := 0.0;
    robot6axis_ctrled1/robot6axis_cams/cam_computation1/linNum AT 5338 : REAL := 0.0;
    robot6axis_ctrled1/robot6axis_cams/cam_computation1/linA AT 5339 : REAL := 0.0;
    robot6axis_ctrled1/robot6axis_cams/cam_computation1/linB AT 5340 : REAL := 0.0;
    robot6axis_ctrled1/robot6axis_cams/cam_computation1/FACTOR AT 5341 : REAL := 1.0;
    robot6axis_ctrled1/robot6axis_cams/cam_profile2/name AT 583 : STRING(50) := 'CamAxis2_exa.txt';
    robot6axis_ctrled1/robot6axis_cams/cam_profile2/nbPoints AT 588 : INT := 0;
    robot6axis_ctrled1/robot6axis_cams/cam_profile2/MasterPoints AT 3048 : ARRAY[1..100] OF REAL := [100(0.0)];
    robot6axis_ctrled1/robot6axis_cams/cam_profile2/SlavePoints AT 3150 : ARRAY[1..100] OF REAL := [100(0.0)];
    robot6axis_ctrled1/robot6axis_cams/cam_profile2/pointer AT 589 : DINT := 0;
    robot6axis_ctrled1/robot6axis_cams/cam_profile2/initialized AT 135 : BOOL := false;
    robot6axis_ctrled1/robot6axis_cams/cam_profile2/pFile AT 616 : DINT := 0;
    robot6axis_ctrled1/robot6axis_cams/cam_profile2/fault_reading AT 136 : BOOL := false;
    robot6axis_ctrled1/robot6axis_cams/cam_profile2/fault_openning AT 137 : BOOL := false;
    robot6axis_ctrled1/robot6axis_cams/cam_profile2/complete_path AT 1203 : STRING(254) := '';
    robot6axis_ctrled1/robot6axis_cams/cam_profile8/name AT 265 : STRING(50) := 'CamAxis2_rej.txt';
    robot6axis_ctrled1/robot6axis_cams/cam_profile8/nbPoints AT 590 : INT := 0;
    robot6axis_ctrled1/robot6axis_cams/cam_profile8/MasterPoints AT 3252 : ARRAY[1..100] OF REAL := [100(0.0)];
    robot6axis_ctrled1/robot6axis_cams/cam_profile8/SlavePoints AT 3354 : ARRAY[1..100] OF REAL := [100(0.0)];
    robot6axis_ctrled1/robot6axis_cams/cam_profile8/pointer AT 591 : DINT := 0;
    robot6axis_ctrled1/robot6axis_cams/cam_profile8/initialized AT 138 : BOOL := false;
    robot6axis_ctrled1/robot6axis_cams/cam_profile8/pFile AT 617 : DINT := 0;
    robot6axis_ctrled1/robot6axis_cams/cam_profile8/fault_reading AT 139 : BOOL := false;
    robot6axis_ctrled1/robot6axis_cams/cam_profile8/fault_openning AT 140 : BOOL := false;
    robot6axis_ctrled1/robot6axis_cams/cam_profile8/complete_path AT 1460 : STRING(254) := '';
    robot6axis_ctrled1/robot6axis_cams/cam_computation2/profileNr AT 524 : DINT := 0;
    robot6axis_ctrled1/robot6axis_cams/cam_computation2/MasterPositionIn AT 18 : REAL := 0.0;
    robot6axis_ctrled1/robot6axis_cams/cam_computation2/nbPoints0 AT 588 : INT := 0;
    robot6axis_ctrled1/robot6axis_cams/cam_computation2/MasterPoints0 AT 3048 : ARRAY[1..100] OF REAL := [100(0.0)];
    robot6axis_ctrled1/robot6axis_cams/cam_computation2/SlavePoints0 AT 3150 : ARRAY[1..100] OF REAL := [100(0.0)];
    robot6axis_ctrled1/robot6axis_cams/cam_computation2/pointer0 AT 589 : DINT := 0;
    robot6axis_ctrled1/robot6axis_cams/cam_computation2/nbPoints1 AT 590 : INT := 0;
    robot6axis_ctrled1/robot6axis_cams/cam_computation2/MasterPoints1 AT 3252 : ARRAY[1..100] OF REAL := [100(0.0)];
    robot6axis_ctrled1/robot6axis_cams/cam_computation2/SlavePoints1 AT 3354 : ARRAY[1..100] OF REAL := [100(0.0)];
    robot6axis_ctrled1/robot6axis_cams/cam_computation2/pointer1 AT 591 : DINT := 0;
    robot6axis_ctrled1/robot6axis_cams/cam_computation2/nbPoints2 AT 577 : INT := 0;
    robot6axis_ctrled1/robot6axis_cams/cam_computation2/MasterPoints2 AT 2116 : ARRAY[1..100] OF REAL := [100(0.0)];
    robot6axis_ctrled1/robot6axis_cams/cam_computation2/SlavePoints2 AT 2014 : ARRAY[1..100] OF REAL := [100(0.0)];
    robot6axis_ctrled1/robot6axis_cams/cam_computation2/pointer2 AT 576 : DINT := 0;
    robot6axis_ctrled1/robot6axis_cams/cam_computation2/nbPoints3 AT 575 : INT := 0;
    robot6axis_ctrled1/robot6axis_cams/cam_computation2/MasterPoints3 AT 1912 : ARRAY[1..100] OF REAL := [100(0.0)];
    robot6axis_ctrled1/robot6axis_cams/cam_computation2/SlavePoints3 AT 1810 : ARRAY[1..100] OF REAL := [100(0.0)];
    robot6axis_ctrled1/robot6axis_cams/cam_computation2/pointer3 AT 574 : DINT := 0;
    robot6axis_ctrled1/robot6axis_cams/cam_computation2/slavePosition AT 168 : REAL := 0.0;
    robot6axis_ctrled1/robot6axis_cams/cam_computation2/masterPosition AT 1809 : REAL := 0.0;
    robot6axis_ctrled1/robot6axis_cams/cam_computation2/i AT 618 : INT := 0;
    robot6axis_ctrled1/robot6axis_cams/cam_computation2/modulo AT 5342 : REAL := 0.0;
    robot6axis_ctrled1/robot6axis_cams/cam_computation2/divider AT 619 : INT := 0;
    robot6axis_ctrled1/robot6axis_cams/cam_computation2/faultProfileNr AT 141 : BOOL := false;
    robot6axis_ctrled1/robot6axis_cams/cam_computation2/faultMasterPositionOOB AT 142 : BOOL := false;
    robot6axis_ctrled1/robot6axis_cams/cam_computation2/faultLinComputation AT 143 : BOOL := false;
    robot6axis_ctrled1/robot6axis_cams/cam_computation2/nbPoints AT 620 : INT := 0;
    robot6axis_ctrled1/robot6axis_cams/cam_computation2/MasterPoints AT 5343 : ARRAY[1..100] OF REAL := [100(0.0)];
    robot6axis_ctrled1/robot6axis_cams/cam_computation2/SlavePoints AT 5445 : ARRAY[1..100] OF REAL := [100(0.0)];
    robot6axis_ctrled1/robot6axis_cams/cam_computation2/found AT 144 : BOOL := false;
    robot6axis_ctrled1/robot6axis_cams/cam_computation2/index AT 621 : INT := 0;
    robot6axis_ctrled1/robot6axis_cams/cam_computation2/linDenom AT 5547 : REAL := 0.0;
    robot6axis_ctrled1/robot6axis_cams/cam_computation2/linNum AT 5548 : REAL := 0.0;
    robot6axis_ctrled1/robot6axis_cams/cam_computation2/linA AT 5549 : REAL := 0.0;
    robot6axis_ctrled1/robot6axis_cams/cam_computation2/linB AT 5550 : REAL := 0.0;
    robot6axis_ctrled1/robot6axis_cams/cam_computation2/FACTOR AT 5551 : REAL := 1.0;
    robot6axis_ctrled1/robot6axis_cams/cam_profile3/name AT 530 : STRING(50) := 'CamAxis3_exa.txt';
    robot6axis_ctrled1/robot6axis_cams/cam_profile3/nbPoints AT 592 : INT := 0;
    robot6axis_ctrled1/robot6axis_cams/cam_profile3/MasterPoints AT 3456 : ARRAY[1..100] OF REAL := [100(0.0)];
    robot6axis_ctrled1/robot6axis_cams/cam_profile3/SlavePoints AT 3558 : ARRAY[1..100] OF REAL := [100(0.0)];
    robot6axis_ctrled1/robot6axis_cams/cam_profile3/pointer AT 593 : DINT := 0;
    robot6axis_ctrled1/robot6axis_cams/cam_profile3/initialized AT 145 : BOOL := false;
    robot6axis_ctrled1/robot6axis_cams/cam_profile3/pFile AT 622 : DINT := 0;
    robot6axis_ctrled1/robot6axis_cams/cam_profile3/fault_reading AT 146 : BOOL := false;
    robot6axis_ctrled1/robot6axis_cams/cam_profile3/fault_openning AT 147 : BOOL := false;
    robot6axis_ctrled1/robot6axis_cams/cam_profile3/complete_path AT 1717 : STRING(254) := '';
    robot6axis_ctrled1/robot6axis_cams/cam_profile9/name AT 212 : STRING(50) := 'CamAxis3_rej.txt';
    robot6axis_ctrled1/robot6axis_cams/cam_profile9/nbPoints AT 594 : INT := 0;
    robot6axis_ctrled1/robot6axis_cams/cam_profile9/MasterPoints AT 3660 : ARRAY[1..100] OF REAL := [100(0.0)];
    robot6axis_ctrled1/robot6axis_cams/cam_profile9/SlavePoints AT 3762 : ARRAY[1..100] OF REAL := [100(0.0)];
    robot6axis_ctrled1/robot6axis_cams/cam_profile9/pointer AT 595 : DINT := 0;
    robot6axis_ctrled1/robot6axis_cams/cam_profile9/initialized AT 148 : BOOL := false;
    robot6axis_ctrled1/robot6axis_cams/cam_profile9/pFile AT 623 : DINT := 0;
    robot6axis_ctrled1/robot6axis_cams/cam_profile9/fault_reading AT 149 : BOOL := false;
    robot6axis_ctrled1/robot6axis_cams/cam_profile9/fault_openning AT 150 : BOOL := false;
    robot6axis_ctrled1/robot6axis_cams/cam_profile9/complete_path AT 1974 : STRING(254) := '';
    robot6axis_ctrled1/robot6axis_cams/cam_computation3/profileNr AT 524 : DINT := 0;
    robot6axis_ctrled1/robot6axis_cams/cam_computation3/MasterPositionIn AT 18 : REAL := 0.0;
    robot6axis_ctrled1/robot6axis_cams/cam_computation3/nbPoints0 AT 592 : INT := 0;
    robot6axis_ctrled1/robot6axis_cams/cam_computation3/MasterPoints0 AT 3456 : ARRAY[1..100] OF REAL := [100(0.0)];
    robot6axis_ctrled1/robot6axis_cams/cam_computation3/SlavePoints0 AT 3558 : ARRAY[1..100] OF REAL := [100(0.0)];
    robot6axis_ctrled1/robot6axis_cams/cam_computation3/pointer0 AT 593 : DINT := 0;
    robot6axis_ctrled1/robot6axis_cams/cam_computation3/nbPoints1 AT 594 : INT := 0;
    robot6axis_ctrled1/robot6axis_cams/cam_computation3/MasterPoints1 AT 3660 : ARRAY[1..100] OF REAL := [100(0.0)];
    robot6axis_ctrled1/robot6axis_cams/cam_computation3/SlavePoints1 AT 3762 : ARRAY[1..100] OF REAL := [100(0.0)];
    robot6axis_ctrled1/robot6axis_cams/cam_computation3/pointer1 AT 595 : DINT := 0;
    robot6axis_ctrled1/robot6axis_cams/cam_computation3/nbPoints2 AT 573 : INT := 0;
    robot6axis_ctrled1/robot6axis_cams/cam_computation3/MasterPoints2 AT 1707 : ARRAY[1..100] OF REAL := [100(0.0)];
    robot6axis_ctrled1/robot6axis_cams/cam_computation3/SlavePoints2 AT 1605 : ARRAY[1..100] OF REAL := [100(0.0)];
    robot6axis_ctrled1/robot6axis_cams/cam_computation3/pointer2 AT 572 : DINT := 0;
    robot6axis_ctrled1/robot6axis_cams/cam_computation3/nbPoints3 AT 571 : INT := 0;
    robot6axis_ctrled1/robot6axis_cams/cam_computation3/MasterPoints3 AT 1503 : ARRAY[1..100] OF REAL := [100(0.0)];
    robot6axis_ctrled1/robot6axis_cams/cam_computation3/SlavePoints3 AT 1401 : ARRAY[1..100] OF REAL := [100(0.0)];
    robot6axis_ctrled1/robot6axis_cams/cam_computation3/pointer3 AT 570 : DINT := 0;
    robot6axis_ctrled1/robot6axis_cams/cam_computation3/slavePosition AT 169 : REAL := 0.0;
    robot6axis_ctrled1/robot6axis_cams/cam_computation3/masterPosition AT 1400 : REAL := 0.0;
    robot6axis_ctrled1/robot6axis_cams/cam_computation3/i AT 624 : INT := 0;
    robot6axis_ctrled1/robot6axis_cams/cam_computation3/modulo AT 5552 : REAL := 0.0;
    robot6axis_ctrled1/robot6axis_cams/cam_computation3/divider AT 625 : INT := 0;
    robot6axis_ctrled1/robot6axis_cams/cam_computation3/faultProfileNr AT 151 : BOOL := false;
    robot6axis_ctrled1/robot6axis_cams/cam_computation3/faultMasterPositionOOB AT 152 : BOOL := false;
    robot6axis_ctrled1/robot6axis_cams/cam_computation3/faultLinComputation AT 153 : BOOL := false;
    robot6axis_ctrled1/robot6axis_cams/cam_computation3/nbPoints AT 626 : INT := 0;
    robot6axis_ctrled1/robot6axis_cams/cam_computation3/MasterPoints AT 5553 : ARRAY[1..100] OF REAL := [100(0.0)];
    robot6axis_ctrled1/robot6axis_cams/cam_computation3/SlavePoints AT 5655 : ARRAY[1..100] OF REAL := [100(0.0)];
    robot6axis_ctrled1/robot6axis_cams/cam_computation3/found AT 154 : BOOL := false;
    robot6axis_ctrled1/robot6axis_cams/cam_computation3/index AT 627 : INT := 0;
    robot6axis_ctrled1/robot6axis_cams/cam_computation3/linDenom AT 5757 : REAL := 0.0;
    robot6axis_ctrled1/robot6axis_cams/cam_computation3/linNum AT 5758 : REAL := 0.0;
    robot6axis_ctrled1/robot6axis_cams/cam_computation3/linA AT 5759 : REAL := 0.0;
    robot6axis_ctrled1/robot6axis_cams/cam_computation3/linB AT 5760 : REAL := 0.0;
    robot6axis_ctrled1/robot6axis_cams/cam_computation3/FACTOR AT 5761 : REAL := 1.0;
    robot6axis_ctrled1/robot6axis_cams/cam_profile4/name AT 477 : STRING(50) := 'CamAxis4_exa.txt';
    robot6axis_ctrled1/robot6axis_cams/cam_profile4/nbPoints AT 596 : INT := 0;
    robot6axis_ctrled1/robot6axis_cams/cam_profile4/MasterPoints AT 3864 : ARRAY[1..100] OF REAL := [100(0.0)];
    robot6axis_ctrled1/robot6axis_cams/cam_profile4/SlavePoints AT 3966 : ARRAY[1..100] OF REAL := [100(0.0)];
    robot6axis_ctrled1/robot6axis_cams/cam_profile4/pointer AT 597 : DINT := 0;
    robot6axis_ctrled1/robot6axis_cams/cam_profile4/initialized AT 155 : BOOL := false;
    robot6axis_ctrled1/robot6axis_cams/cam_profile4/pFile AT 628 : DINT := 0;
    robot6axis_ctrled1/robot6axis_cams/cam_profile4/fault_reading AT 156 : BOOL := false;
    robot6axis_ctrled1/robot6axis_cams/cam_profile4/fault_openning AT 157 : BOOL := false;
    robot6axis_ctrled1/robot6axis_cams/cam_profile4/complete_path AT 2231 : STRING(254) := '';
    robot6axis_ctrled1/robot6axis_cams/cam_profile10/name AT 159 : STRING(50) := 'CamAxis4_rej.txt';
    robot6axis_ctrled1/robot6axis_cams/cam_profile10/nbPoints AT 598 : INT := 0;
    robot6axis_ctrled1/robot6axis_cams/cam_profile10/MasterPoints AT 4068 : ARRAY[1..100] OF REAL := [100(0.0)];
    robot6axis_ctrled1/robot6axis_cams/cam_profile10/SlavePoints AT 4170 : ARRAY[1..100] OF REAL := [100(0.0)];
    robot6axis_ctrled1/robot6axis_cams/cam_profile10/pointer AT 599 : DINT := 0;
    robot6axis_ctrled1/robot6axis_cams/cam_profile10/initialized AT 158 : BOOL := false;
    robot6axis_ctrled1/robot6axis_cams/cam_profile10/pFile AT 629 : DINT := 0;
    robot6axis_ctrled1/robot6axis_cams/cam_profile10/fault_reading AT 159 : BOOL := false;
    robot6axis_ctrled1/robot6axis_cams/cam_profile10/fault_openning AT 160 : BOOL := false;
    robot6axis_ctrled1/robot6axis_cams/cam_profile10/complete_path AT 2488 : STRING(254) := '';
    robot6axis_ctrled1/robot6axis_cams/cam_computation4/profileNr AT 524 : DINT := 0;
    robot6axis_ctrled1/robot6axis_cams/cam_computation4/MasterPositionIn AT 18 : REAL := 0.0;
    robot6axis_ctrled1/robot6axis_cams/cam_computation4/nbPoints0 AT 596 : INT := 0;
    robot6axis_ctrled1/robot6axis_cams/cam_computation4/MasterPoints0 AT 3864 : ARRAY[1..100] OF REAL := [100(0.0)];
    robot6axis_ctrled1/robot6axis_cams/cam_computation4/SlavePoints0 AT 3966 : ARRAY[1..100] OF REAL := [100(0.0)];
    robot6axis_ctrled1/robot6axis_cams/cam_computation4/pointer0 AT 597 : DINT := 0;
    robot6axis_ctrled1/robot6axis_cams/cam_computation4/nbPoints1 AT 598 : INT := 0;
    robot6axis_ctrled1/robot6axis_cams/cam_computation4/MasterPoints1 AT 4068 : ARRAY[1..100] OF REAL := [100(0.0)];
    robot6axis_ctrled1/robot6axis_cams/cam_computation4/SlavePoints1 AT 4170 : ARRAY[1..100] OF REAL := [100(0.0)];
    robot6axis_ctrled1/robot6axis_cams/cam_computation4/pointer1 AT 599 : DINT := 0;
    robot6axis_ctrled1/robot6axis_cams/cam_computation4/nbPoints2 AT 569 : INT := 0;
    robot6axis_ctrled1/robot6axis_cams/cam_computation4/MasterPoints2 AT 1298 : ARRAY[1..100] OF REAL := [100(0.0)];
    robot6axis_ctrled1/robot6axis_cams/cam_computation4/SlavePoints2 AT 1196 : ARRAY[1..100] OF REAL := [100(0.0)];
    robot6axis_ctrled1/robot6axis_cams/cam_computation4/pointer2 AT 568 : DINT := 0;
    robot6axis_ctrled1/robot6axis_cams/cam_computation4/nbPoints3 AT 567 : INT := 0;
    robot6axis_ctrled1/robot6axis_cams/cam_computation4/MasterPoints3 AT 1094 : ARRAY[1..100] OF REAL := [100(0.0)];
    robot6axis_ctrled1/robot6axis_cams/cam_computation4/SlavePoints3 AT 992 : ARRAY[1..100] OF REAL := [100(0.0)];
    robot6axis_ctrled1/robot6axis_cams/cam_computation4/pointer3 AT 566 : DINT := 0;
    robot6axis_ctrled1/robot6axis_cams/cam_computation4/slavePosition AT 170 : REAL := 0.0;
    robot6axis_ctrled1/robot6axis_cams/cam_computation4/masterPosition AT 991 : REAL := 0.0;
    robot6axis_ctrled1/robot6axis_cams/cam_computation4/i AT 630 : INT := 0;
    robot6axis_ctrled1/robot6axis_cams/cam_computation4/modulo AT 5762 : REAL := 0.0;
    robot6axis_ctrled1/robot6axis_cams/cam_computation4/divider AT 631 : INT := 0;
    robot6axis_ctrled1/robot6axis_cams/cam_computation4/faultProfileNr AT 161 : BOOL := false;
    robot6axis_ctrled1/robot6axis_cams/cam_computation4/faultMasterPositionOOB AT 162 : BOOL := false;
    robot6axis_ctrled1/robot6axis_cams/cam_computation4/faultLinComputation AT 163 : BOOL := false;
    robot6axis_ctrled1/robot6axis_cams/cam_computation4/nbPoints AT 632 : INT := 0;
    robot6axis_ctrled1/robot6axis_cams/cam_computation4/MasterPoints AT 5763 : ARRAY[1..100] OF REAL := [100(0.0)];
    robot6axis_ctrled1/robot6axis_cams/cam_computation4/SlavePoints AT 5865 : ARRAY[1..100] OF REAL := [100(0.0)];
    robot6axis_ctrled1/robot6axis_cams/cam_computation4/found AT 164 : BOOL := false;
    robot6axis_ctrled1/robot6axis_cams/cam_computation4/index AT 633 : INT := 0;
    robot6axis_ctrled1/robot6axis_cams/cam_computation4/linDenom AT 5967 : REAL := 0.0;
    robot6axis_ctrled1/robot6axis_cams/cam_computation4/linNum AT 5968 : REAL := 0.0;
    robot6axis_ctrled1/robot6axis_cams/cam_computation4/linA AT 5969 : REAL := 0.0;
    robot6axis_ctrled1/robot6axis_cams/cam_computation4/linB AT 5970 : REAL := 0.0;
    robot6axis_ctrled1/robot6axis_cams/cam_computation4/FACTOR AT 5971 : REAL := 1.0;
    robot6axis_ctrled1/robot6axis_cams/cam_profile5/name AT 424 : STRING(50) := 'CamAxis5_exa.txt';
    robot6axis_ctrled1/robot6axis_cams/cam_profile5/nbPoints AT 600 : INT := 0;
    robot6axis_ctrled1/robot6axis_cams/cam_profile5/MasterPoints AT 4272 : ARRAY[1..100] OF REAL := [100(0.0)];
    robot6axis_ctrled1/robot6axis_cams/cam_profile5/SlavePoints AT 4374 : ARRAY[1..100] OF REAL := [100(0.0)];
    robot6axis_ctrled1/robot6axis_cams/cam_profile5/pointer AT 601 : DINT := 0;
    robot6axis_ctrled1/robot6axis_cams/cam_profile5/initialized AT 165 : BOOL := false;
    robot6axis_ctrled1/robot6axis_cams/cam_profile5/pFile AT 634 : DINT := 0;
    robot6axis_ctrled1/robot6axis_cams/cam_profile5/fault_reading AT 166 : BOOL := false;
    robot6axis_ctrled1/robot6axis_cams/cam_profile5/fault_openning AT 167 : BOOL := false;
    robot6axis_ctrled1/robot6axis_cams/cam_profile5/complete_path AT 2745 : STRING(254) := '';
    robot6axis_ctrled1/robot6axis_cams/cam_profile11/name AT 106 : STRING(50) := 'CamAxis5_rej.txt';
    robot6axis_ctrled1/robot6axis_cams/cam_profile11/nbPoints AT 602 : INT := 0;
    robot6axis_ctrled1/robot6axis_cams/cam_profile11/MasterPoints AT 4476 : ARRAY[1..100] OF REAL := [100(0.0)];
    robot6axis_ctrled1/robot6axis_cams/cam_profile11/SlavePoints AT 4578 : ARRAY[1..100] OF REAL := [100(0.0)];
    robot6axis_ctrled1/robot6axis_cams/cam_profile11/pointer AT 603 : DINT := 0;
    robot6axis_ctrled1/robot6axis_cams/cam_profile11/initialized AT 168 : BOOL := false;
    robot6axis_ctrled1/robot6axis_cams/cam_profile11/pFile AT 635 : DINT := 0;
    robot6axis_ctrled1/robot6axis_cams/cam_profile11/fault_reading AT 169 : BOOL := false;
    robot6axis_ctrled1/robot6axis_cams/cam_profile11/fault_openning AT 170 : BOOL := false;
    robot6axis_ctrled1/robot6axis_cams/cam_profile11/complete_path AT 3002 : STRING(254) := '';
    robot6axis_ctrled1/robot6axis_cams/cam_computation5/profileNr AT 524 : DINT := 0;
    robot6axis_ctrled1/robot6axis_cams/cam_computation5/MasterPositionIn AT 18 : REAL := 0.0;
    robot6axis_ctrled1/robot6axis_cams/cam_computation5/nbPoints0 AT 600 : INT := 0;
    robot6axis_ctrled1/robot6axis_cams/cam_computation5/MasterPoints0 AT 4272 : ARRAY[1..100] OF REAL := [100(0.0)];
    robot6axis_ctrled1/robot6axis_cams/cam_computation5/SlavePoints0 AT 4374 : ARRAY[1..100] OF REAL := [100(0.0)];
    robot6axis_ctrled1/robot6axis_cams/cam_computation5/pointer0 AT 601 : DINT := 0;
    robot6axis_ctrled1/robot6axis_cams/cam_computation5/nbPoints1 AT 602 : INT := 0;
    robot6axis_ctrled1/robot6axis_cams/cam_computation5/MasterPoints1 AT 4476 : ARRAY[1..100] OF REAL := [100(0.0)];
    robot6axis_ctrled1/robot6axis_cams/cam_computation5/SlavePoints1 AT 4578 : ARRAY[1..100] OF REAL := [100(0.0)];
    robot6axis_ctrled1/robot6axis_cams/cam_computation5/pointer1 AT 603 : DINT := 0;
    robot6axis_ctrled1/robot6axis_cams/cam_computation5/nbPoints2 AT 565 : INT := 0;
    robot6axis_ctrled1/robot6axis_cams/cam_computation5/MasterPoints2 AT 889 : ARRAY[1..100] OF REAL := [100(0.0)];
    robot6axis_ctrled1/robot6axis_cams/cam_computation5/SlavePoints2 AT 787 : ARRAY[1..100] OF REAL := [100(0.0)];
    robot6axis_ctrled1/robot6axis_cams/cam_computation5/pointer2 AT 564 : DINT := 0;
    robot6axis_ctrled1/robot6axis_cams/cam_computation5/nbPoints3 AT 563 : INT := 0;
    robot6axis_ctrled1/robot6axis_cams/cam_computation5/MasterPoints3 AT 685 : ARRAY[1..100] OF REAL := [100(0.0)];
    robot6axis_ctrled1/robot6axis_cams/cam_computation5/SlavePoints3 AT 583 : ARRAY[1..100] OF REAL := [100(0.0)];
    robot6axis_ctrled1/robot6axis_cams/cam_computation5/pointer3 AT 562 : DINT := 0;
    robot6axis_ctrled1/robot6axis_cams/cam_computation5/slavePosition AT 171 : REAL := 0.0;
    robot6axis_ctrled1/robot6axis_cams/cam_computation5/masterPosition AT 582 : REAL := 0.0;
    robot6axis_ctrled1/robot6axis_cams/cam_computation5/i AT 636 : INT := 0;
    robot6axis_ctrled1/robot6axis_cams/cam_computation5/modulo AT 5972 : REAL := 0.0;
    robot6axis_ctrled1/robot6axis_cams/cam_computation5/divider AT 637 : INT := 0;
    robot6axis_ctrled1/robot6axis_cams/cam_computation5/faultProfileNr AT 171 : BOOL := false;
    robot6axis_ctrled1/robot6axis_cams/cam_computation5/faultMasterPositionOOB AT 172 : BOOL := false;
    robot6axis_ctrled1/robot6axis_cams/cam_computation5/faultLinComputation AT 173 : BOOL := false;
    robot6axis_ctrled1/robot6axis_cams/cam_computation5/nbPoints AT 638 : INT := 0;
    robot6axis_ctrled1/robot6axis_cams/cam_computation5/MasterPoints AT 5973 : ARRAY[1..100] OF REAL := [100(0.0)];
    robot6axis_ctrled1/robot6axis_cams/cam_computation5/SlavePoints AT 6075 : ARRAY[1..100] OF REAL := [100(0.0)];
    robot6axis_ctrled1/robot6axis_cams/cam_computation5/found AT 174 : BOOL := false;
    robot6axis_ctrled1/robot6axis_cams/cam_computation5/index AT 639 : INT := 0;
    robot6axis_ctrled1/robot6axis_cams/cam_computation5/linDenom AT 6177 : REAL := 0.0;
    robot6axis_ctrled1/robot6axis_cams/cam_computation5/linNum AT 6178 : REAL := 0.0;
    robot6axis_ctrled1/robot6axis_cams/cam_computation5/linA AT 6179 : REAL := 0.0;
    robot6axis_ctrled1/robot6axis_cams/cam_computation5/linB AT 6180 : REAL := 0.0;
    robot6axis_ctrled1/robot6axis_cams/cam_computation5/FACTOR AT 6181 : REAL := 1.0;
    robot6axis_ctrled1/robot6axis_cams/cam_profile6/name AT 371 : STRING(50) := 'CamAxis6_exa.txt';
    robot6axis_ctrled1/robot6axis_cams/cam_profile6/nbPoints AT 604 : INT := 0;
    robot6axis_ctrled1/robot6axis_cams/cam_profile6/MasterPoints AT 4680 : ARRAY[1..100] OF REAL := [100(0.0)];
    robot6axis_ctrled1/robot6axis_cams/cam_profile6/SlavePoints AT 4782 : ARRAY[1..100] OF REAL := [100(0.0)];
    robot6axis_ctrled1/robot6axis_cams/cam_profile6/pointer AT 605 : DINT := 0;
    robot6axis_ctrled1/robot6axis_cams/cam_profile6/initialized AT 175 : BOOL := false;
    robot6axis_ctrled1/robot6axis_cams/cam_profile6/pFile AT 640 : DINT := 0;
    robot6axis_ctrled1/robot6axis_cams/cam_profile6/fault_reading AT 176 : BOOL := false;
    robot6axis_ctrled1/robot6axis_cams/cam_profile6/fault_openning AT 177 : BOOL := false;
    robot6axis_ctrled1/robot6axis_cams/cam_profile6/complete_path AT 3259 : STRING(254) := '';
    robot6axis_ctrled1/robot6axis_cams/cam_profile12/name AT 53 : STRING(50) := 'CamAxis6_rej.txt';
    robot6axis_ctrled1/robot6axis_cams/cam_profile12/nbPoints AT 606 : INT := 0;
    robot6axis_ctrled1/robot6axis_cams/cam_profile12/MasterPoints AT 4884 : ARRAY[1..100] OF REAL := [100(0.0)];
    robot6axis_ctrled1/robot6axis_cams/cam_profile12/SlavePoints AT 4986 : ARRAY[1..100] OF REAL := [100(0.0)];
    robot6axis_ctrled1/robot6axis_cams/cam_profile12/pointer AT 607 : DINT := 0;
    robot6axis_ctrled1/robot6axis_cams/cam_profile12/initialized AT 178 : BOOL := false;
    robot6axis_ctrled1/robot6axis_cams/cam_profile12/pFile AT 641 : DINT := 0;
    robot6axis_ctrled1/robot6axis_cams/cam_profile12/fault_reading AT 179 : BOOL := false;
    robot6axis_ctrled1/robot6axis_cams/cam_profile12/fault_openning AT 180 : BOOL := false;
    robot6axis_ctrled1/robot6axis_cams/cam_profile12/complete_path AT 3516 : STRING(254) := '';
    robot6axis_ctrled1/robot6axis_cams/cam_computation6/profileNr AT 524 : DINT := 0;
    robot6axis_ctrled1/robot6axis_cams/cam_computation6/MasterPositionIn AT 18 : REAL := 0.0;
    robot6axis_ctrled1/robot6axis_cams/cam_computation6/nbPoints0 AT 604 : INT := 0;
    robot6axis_ctrled1/robot6axis_cams/cam_computation6/MasterPoints0 AT 4680 : ARRAY[1..100] OF REAL := [100(0.0)];
    robot6axis_ctrled1/robot6axis_cams/cam_computation6/SlavePoints0 AT 4782 : ARRAY[1..100] OF REAL := [100(0.0)];
    robot6axis_ctrled1/robot6axis_cams/cam_computation6/pointer0 AT 605 : DINT := 0;
    robot6axis_ctrled1/robot6axis_cams/cam_computation6/nbPoints1 AT 606 : INT := 0;
    robot6axis_ctrled1/robot6axis_cams/cam_computation6/MasterPoints1 AT 4884 : ARRAY[1..100] OF REAL := [100(0.0)];
    robot6axis_ctrled1/robot6axis_cams/cam_computation6/SlavePoints1 AT 4986 : ARRAY[1..100] OF REAL := [100(0.0)];
    robot6axis_ctrled1/robot6axis_cams/cam_computation6/pointer1 AT 607 : DINT := 0;
    robot6axis_ctrled1/robot6axis_cams/cam_computation6/nbPoints2 AT 561 : INT := 0;
    robot6axis_ctrled1/robot6axis_cams/cam_computation6/MasterPoints2 AT 480 : ARRAY[1..100] OF REAL := [100(0.0)];
    robot6axis_ctrled1/robot6axis_cams/cam_computation6/SlavePoints2 AT 378 : ARRAY[1..100] OF REAL := [100(0.0)];
    robot6axis_ctrled1/robot6axis_cams/cam_computation6/pointer2 AT 560 : DINT := 0;
    robot6axis_ctrled1/robot6axis_cams/cam_computation6/nbPoints3 AT 559 : INT := 0;
    robot6axis_ctrled1/robot6axis_cams/cam_computation6/MasterPoints3 AT 276 : ARRAY[1..100] OF REAL := [100(0.0)];
    robot6axis_ctrled1/robot6axis_cams/cam_computation6/SlavePoints3 AT 174 : ARRAY[1..100] OF REAL := [100(0.0)];
    robot6axis_ctrled1/robot6axis_cams/cam_computation6/pointer3 AT 558 : DINT := 0;
    robot6axis_ctrled1/robot6axis_cams/cam_computation6/slavePosition AT 172 : REAL := 0.0;
    robot6axis_ctrled1/robot6axis_cams/cam_computation6/masterPosition AT 173 : REAL := 0.0;
    robot6axis_ctrled1/robot6axis_cams/cam_computation6/i AT 642 : INT := 0;
    robot6axis_ctrled1/robot6axis_cams/cam_computation6/modulo AT 6182 : REAL := 0.0;
    robot6axis_ctrled1/robot6axis_cams/cam_computation6/divider AT 643 : INT := 0;
    robot6axis_ctrled1/robot6axis_cams/cam_computation6/faultProfileNr AT 181 : BOOL := false;
    robot6axis_ctrled1/robot6axis_cams/cam_computation6/faultMasterPositionOOB AT 182 : BOOL := false;
    robot6axis_ctrled1/robot6axis_cams/cam_computation6/faultLinComputation AT 183 : BOOL := false;
    robot6axis_ctrled1/robot6axis_cams/cam_computation6/nbPoints AT 644 : INT := 0;
    robot6axis_ctrled1/robot6axis_cams/cam_computation6/MasterPoints AT 6183 : ARRAY[1..100] OF REAL := [100(0.0)];
    robot6axis_ctrled1/robot6axis_cams/cam_computation6/SlavePoints AT 6285 : ARRAY[1..100] OF REAL := [100(0.0)];
    robot6axis_ctrled1/robot6axis_cams/cam_computation6/found AT 184 : BOOL := false;
    robot6axis_ctrled1/robot6axis_cams/cam_computation6/index AT 645 : INT := 0;
    robot6axis_ctrled1/robot6axis_cams/cam_computation6/linDenom AT 6387 : REAL := 0.0;
    robot6axis_ctrled1/robot6axis_cams/cam_computation6/linNum AT 6388 : REAL := 0.0;
    robot6axis_ctrled1/robot6axis_cams/cam_computation6/linA AT 6389 : REAL := 0.0;
    robot6axis_ctrled1/robot6axis_cams/cam_computation6/linB AT 6390 : REAL := 0.0;
    robot6axis_ctrled1/robot6axis_cams/cam_computation6/FACTOR AT 6391 : REAL := 1.0;
    robot6axis_ctrled1/robot6axis/armOrigin AT 27 : ARRAY[1..3] OF REAL := [800.0, 400.0, 0.0];
    robot6axis_ctrled1/robot6axis/structRotVectorFOOT AT 162 : ARRAY[1..3] OF REAL := [0.0, 1.0, 0.0];
    robot6axis_ctrled1/robot6axis/structRotDegFOOT AT 161 : REAL := -90.01;
    robot6axis_ctrled1/robot6axis/ownRotDegFOOT AT 160 : REAL := 90.0;
    robot6axis_ctrled1/robot6axis/structRotVectorFOOT2 AT 155 : ARRAY[1..3] OF REAL := [2(0.0), 1.0];
    robot6axis_ctrled1/robot6axis/structRotDegFOOT2 AT 154 : REAL := 90.0;
    robot6axis_ctrled1/robot6axis/structRotVectorArm2 AT 149 : ARRAY[1..3] OF REAL := [2(0.0), 1.0];
    robot6axis_ctrled1/robot6axis/structRotDegArm2 AT 148 : REAL := -90.0;
    robot6axis_ctrled1/robot6axis/driveRotVector1 AT 143 : ARRAY[1..3] OF REAL := [1.0, 2(0.0)];
    robot6axis_ctrled1/robot6axis/driveRotVector2 AT 138 : ARRAY[1..3] OF REAL := [0.0, 1.0, 0.0];
    robot6axis_ctrled1/robot6axis/driveRotVector3 AT 133 : ARRAY[1..3] OF REAL := [0.0, 1.0, 0.0];
    robot6axis_ctrled1/robot6axis/driveRotVector4 AT 128 : ARRAY[1..3] OF REAL := [1.0, 2(0.0)];
    robot6axis_ctrled1/robot6axis/driveRotVector5 AT 123 : ARRAY[1..3] OF REAL := [0.0, 1.0, 0.0];
    robot6axis_ctrled1/robot6axis/driveRotVector6 AT 118 : ARRAY[1..3] OF REAL := [1.0, 2(0.0)];
    robot6axis_ctrled1/robot6axis/structRotVector1RowA AT 113 : ARRAY[1..3] OF REAL := [0.0, 1.0, 0.0];
    robot6axis_ctrled1/robot6axis/structRotDeg1RowA AT 112 : REAL := -90.0;
    robot6axis_ctrled1/robot6axis/structRotVector1RowB AT 107 : ARRAY[1..3] OF REAL := [0.0, 1.0, 0.0];
    robot6axis_ctrled1/robot6axis/structRotDeg1RowB AT 106 : REAL := 90.0;
    robot6axis_ctrled1/robot6axis/structRotVectorMultiRowsA AT 101 : ARRAY[1..3] OF REAL := [0.0, 1.0, 0.0];
    robot6axis_ctrled1/robot6axis/structRotDegMultiRowsA AT 100 : REAL := 90.0;
    robot6axis_ctrled1/robot6axis/structRotVectorMultiRowsB AT 95 : ARRAY[1..3] OF REAL := [0.0, 1.0, 0.0];
    robot6axis_ctrled1/robot6axis/structRotDegMultiRowsB AT 94 : REAL := -90.0;
    robot6axis_ctrled1/robot6axis/HomeCmd AT 98 : BOOL := false;
    robot6axis_ctrled1/robot6axis/MoveVelCmd AT 97 : BOOL := false;
    robot6axis_ctrled1/robot6axis/MoveAbsCmd AT 96 : BOOL := false;
    robot6axis_ctrled1/robot6axis/MoveVel1ManualCmd AT 95 : BOOL := false;
    robot6axis_ctrled1/robot6axis/MoveVel2ManualCmd AT 94 : BOOL := false;
    robot6axis_ctrled1/robot6axis/MoveAbs1ManualCmd AT 93 : BOOL := false;
    robot6axis_ctrled1/robot6axis/MoveAbs2ManualCmd AT 92 : BOOL := false;
    robot6axis_ctrled1/robot6axis/StopCmd AT 22 : BOOL := false;
    robot6axis_ctrled1/robot6axis/MovePosition AT 93 : REAL := 0.0;
    robot6axis_ctrled1/robot6axis/MoveSpeed AT 92 : REAL := 100.0;
    robot6axis_ctrled1/robot6axis/MoveAcceleration AT 91 : REAL := 100.0;
    robot6axis_ctrled1/robot6axis/MoveDeceleration AT 90 : REAL := 100.0;
    robot6axis_ctrled1/robot6axis/offsetAxToMa AT 89 : REAL := 0.0;
    robot6axis_ctrled1/robot6axis/HomeCmd2 AT 91 : BOOL := false;
    robot6axis_ctrled1/robot6axis/MoveVelCmd2 AT 90 : BOOL := false;
    robot6axis_ctrled1/robot6axis/MoveAbsCmd2 AT 89 : BOOL := false;
    robot6axis_ctrled1/robot6axis/MoveVel1ManualCmd2 AT 88 : BOOL := false;
    robot6axis_ctrled1/robot6axis/MoveVel2ManualCmd2 AT 87 : BOOL := false;
    robot6axis_ctrled1/robot6axis/MoveAbs1ManualCmd2 AT 86 : BOOL := false;
    robot6axis_ctrled1/robot6axis/MoveAbs2ManualCmd2 AT 85 : BOOL := false;
    robot6axis_ctrled1/robot6axis/StopCmd2 AT 22 : BOOL := false;
    robot6axis_ctrled1/robot6axis/MovePosition2 AT 88 : REAL := 0.0;
    robot6axis_ctrled1/robot6axis/MoveSpeed2 AT 87 : REAL := 100.0;
    robot6axis_ctrled1/robot6axis/MoveAcceleration2 AT 86 : REAL := 100.0;
    robot6axis_ctrled1/robot6axis/MoveDeceleration2 AT 85 : REAL := 100.0;
    robot6axis_ctrled1/robot6axis/offsetAxToMa2 AT 84 : REAL := 0.0;
    robot6axis_ctrled1/robot6axis/HomeCmd3 AT 84 : BOOL := false;
    robot6axis_ctrled1/robot6axis/MoveVelCmd3 AT 83 : BOOL := false;
    robot6axis_ctrled1/robot6axis/MoveAbsCmd3 AT 82 : BOOL := false;
    robot6axis_ctrled1/robot6axis/MoveVel1ManualCmd3 AT 81 : BOOL := false;
    robot6axis_ctrled1/robot6axis/MoveVel2ManualCmd3 AT 80 : BOOL := false;
    robot6axis_ctrled1/robot6axis/MoveAbs1ManualCmd3 AT 79 : BOOL := false;
    robot6axis_ctrled1/robot6axis/MoveAbs2ManualCmd3 AT 78 : BOOL := false;
    robot6axis_ctrled1/robot6axis/StopCmd3 AT 22 : BOOL := false;
    robot6axis_ctrled1/robot6axis/MovePosition3 AT 83 : REAL := 0.0;
    robot6axis_ctrled1/robot6axis/MoveSpeed3 AT 82 : REAL := 100.0;
    robot6axis_ctrled1/robot6axis/MoveAcceleration3 AT 81 : REAL := 100.0;
    robot6axis_ctrled1/robot6axis/MoveDeceleration3 AT 80 : REAL := 100.0;
    robot6axis_ctrled1/robot6axis/offsetAxToMa3 AT 79 : REAL := 0.0;
    robot6axis_ctrled1/robot6axis/HomeCmd4 AT 77 : BOOL := false;
    robot6axis_ctrled1/robot6axis/MoveVelCmd4 AT 76 : BOOL := false;
    robot6axis_ctrled1/robot6axis/MoveAbsCmd4 AT 75 : BOOL := false;
    robot6axis_ctrled1/robot6axis/MoveVel1ManualCmd4 AT 74 : BOOL := false;
    robot6axis_ctrled1/robot6axis/MoveVel2ManualCmd4 AT 73 : BOOL := false;
    robot6axis_ctrled1/robot6axis/MoveAbs1ManualCmd4 AT 72 : BOOL := false;
    robot6axis_ctrled1/robot6axis/MoveAbs2ManualCmd4 AT 71 : BOOL := false;
    robot6axis_ctrled1/robot6axis/StopCmd4 AT 22 : BOOL := false;
    robot6axis_ctrled1/robot6axis/MovePosition4 AT 78 : REAL := 0.0;
    robot6axis_ctrled1/robot6axis/MoveSpeed4 AT 77 : REAL := 100.0;
    robot6axis_ctrled1/robot6axis/MoveAcceleration4 AT 76 : REAL := 100.0;
    robot6axis_ctrled1/robot6axis/MoveDeceleration4 AT 75 : REAL := 100.0;
    robot6axis_ctrled1/robot6axis/offsetAxToMa4 AT 74 : REAL := 0.0;
    robot6axis_ctrled1/robot6axis/HomeCmd5 AT 70 : BOOL := false;
    robot6axis_ctrled1/robot6axis/MoveVelCmd5 AT 69 : BOOL := false;
    robot6axis_ctrled1/robot6axis/MoveAbsCmd5 AT 68 : BOOL := false;
    robot6axis_ctrled1/robot6axis/MoveVel1ManualCmd5 AT 67 : BOOL := false;
    robot6axis_ctrled1/robot6axis/MoveVel2ManualCmd5 AT 66 : BOOL := false;
    robot6axis_ctrled1/robot6axis/MoveAbs1ManualCmd5 AT 65 : BOOL := false;
    robot6axis_ctrled1/robot6axis/MoveAbs2ManualCmd5 AT 64 : BOOL := false;
    robot6axis_ctrled1/robot6axis/StopCmd5 AT 22 : BOOL := false;
    robot6axis_ctrled1/robot6axis/MovePosition5 AT 73 : REAL := 0.0;
    robot6axis_ctrled1/robot6axis/MoveSpeed5 AT 72 : REAL := 100.0;
    robot6axis_ctrled1/robot6axis/MoveAcceleration5 AT 71 : REAL := 100.0;
    robot6axis_ctrled1/robot6axis/MoveDeceleration5 AT 70 : REAL := 100.0;
    robot6axis_ctrled1/robot6axis/offsetAxToMa5 AT 69 : REAL := 0.0;
    robot6axis_ctrled1/robot6axis/HomeCmd6 AT 63 : BOOL := false;
    robot6axis_ctrled1/robot6axis/MoveVelCmd6 AT 62 : BOOL := false;
    robot6axis_ctrled1/robot6axis/MoveAbsCmd6 AT 61 : BOOL := false;
    robot6axis_ctrled1/robot6axis/MoveVel1ManualCmd6 AT 60 : BOOL := false;
    robot6axis_ctrled1/robot6axis/MoveVel2ManualCmd6 AT 59 : BOOL := false;
    robot6axis_ctrled1/robot6axis/MoveAbs1ManualCmd6 AT 58 : BOOL := false;
    robot6axis_ctrled1/robot6axis/MoveAbs2ManualCmd6 AT 57 : BOOL := false;
    robot6axis_ctrled1/robot6axis/StopCmd6 AT 22 : BOOL := false;
    robot6axis_ctrled1/robot6axis/MovePosition6 AT 68 : REAL := 0.0;
    robot6axis_ctrled1/robot6axis/MoveSpeed6 AT 67 : REAL := 100.0;
    robot6axis_ctrled1/robot6axis/MoveAcceleration6 AT 66 : REAL := 100.0;
    robot6axis_ctrled1/robot6axis/MoveDeceleration6 AT 65 : REAL := 100.0;
    robot6axis_ctrled1/robot6axis/offsetAxToMa6 AT 64 : REAL := 0.0;
    robot6axis_ctrled1/robot6axis/PLC_StatusReady AT 56 : BOOL := true;
    robot6axis_ctrled1/robot6axis/PLC_StatusMoved AT 55 : BOOL := false;
    robot6axis_ctrled1/robot6axis/PLC_StatusStand AT 54 : BOOL := false;
    robot6axis_ctrled1/robot6axis/PLC_ActualPositionAx AT 167 : REAL := 0.0;
    robot6axis_ctrled1/robot6axis/PLC_ActualPositionMa AT 63 : REAL := 0.0;
    robot6axis_ctrled1/robot6axis/PLC_ActualVelocity AT 62 : REAL := 0.0;
    robot6axis_ctrled1/robot6axis/PLC_StatusReady2 AT 53 : BOOL := true;
    robot6axis_ctrled1/robot6axis/PLC_StatusMoved2 AT 52 : BOOL := false;
    robot6axis_ctrled1/robot6axis/PLC_StatusStand2 AT 51 : BOOL := false;
    robot6axis_ctrled1/robot6axis/PLC_ActualPositionAx2 AT 168 : REAL := 0.0;
    robot6axis_ctrled1/robot6axis/PLC_ActualPositionMa2 AT 61 : REAL := 0.0;
    robot6axis_ctrled1/robot6axis/PLC_ActualVelocity2 AT 60 : REAL := 0.0;
    robot6axis_ctrled1/robot6axis/PLC_StatusReady3 AT 50 : BOOL := true;
    robot6axis_ctrled1/robot6axis/PLC_StatusMoved3 AT 49 : BOOL := false;
    robot6axis_ctrled1/robot6axis/PLC_StatusStand3 AT 48 : BOOL := false;
    robot6axis_ctrled1/robot6axis/PLC_ActualPositionAx3 AT 169 : REAL := 0.0;
    robot6axis_ctrled1/robot6axis/PLC_ActualPositionMa3 AT 59 : REAL := 0.0;
    robot6axis_ctrled1/robot6axis/PLC_ActualVelocity3 AT 58 : REAL := 0.0;
    robot6axis_ctrled1/robot6axis/PLC_StatusReady4 AT 47 : BOOL := true;
    robot6axis_ctrled1/robot6axis/PLC_StatusMoved4 AT 46 : BOOL := false;
    robot6axis_ctrled1/robot6axis/PLC_StatusStand4 AT 45 : BOOL := false;
    robot6axis_ctrled1/robot6axis/PLC_ActualPositionAx4 AT 170 : REAL := 0.0;
    robot6axis_ctrled1/robot6axis/PLC_ActualPositionMa4 AT 57 : REAL := 0.0;
    robot6axis_ctrled1/robot6axis/PLC_ActualVelocity4 AT 56 : REAL := 0.0;
    robot6axis_ctrled1/robot6axis/PLC_StatusReady5 AT 44 : BOOL := true;
    robot6axis_ctrled1/robot6axis/PLC_StatusMoved5 AT 43 : BOOL := false;
    robot6axis_ctrled1/robot6axis/PLC_StatusStand5 AT 42 : BOOL := false;
    robot6axis_ctrled1/robot6axis/PLC_ActualPositionAx5 AT 171 : REAL := 0.0;
    robot6axis_ctrled1/robot6axis/PLC_ActualPositionMa5 AT 55 : REAL := 0.0;
    robot6axis_ctrled1/robot6axis/PLC_ActualVelocity5 AT 54 : REAL := 0.0;
    robot6axis_ctrled1/robot6axis/PLC_StatusReady6 AT 41 : BOOL := true;
    robot6axis_ctrled1/robot6axis/PLC_StatusMoved6 AT 40 : BOOL := false;
    robot6axis_ctrled1/robot6axis/PLC_StatusStand6 AT 39 : BOOL := false;
    robot6axis_ctrled1/robot6axis/PLC_ActualPositionAx6 AT 172 : REAL := 0.0;
    robot6axis_ctrled1/robot6axis/PLC_ActualPositionMa6 AT 53 : REAL := 0.0;
    robot6axis_ctrled1/robot6axis/PLC_ActualVelocity6 AT 52 : REAL := 0.0;
    robot6axis_ctrled1/robot6axis/gripSyringes AT 21 : BOOL := false;
    robot6axis_ctrled1/robot6axis/ActualVelocity1 AT 51 : REAL := 0.0;
    robot6axis_ctrled1/robot6axis/ActualVelocity2 AT 50 : REAL := 0.0;
    robot6axis_ctrled1/robot6axis/ActualVelocity3 AT 49 : REAL := 0.0;
    robot6axis_ctrled1/robot6axis/ActualVelocity4 AT 48 : REAL := 0.0;
    robot6axis_ctrled1/robot6axis/ActualVelocity5 AT 47 : REAL := 0.0;
    robot6axis_ctrled1/robot6axis/ActualVelocity6 AT 46 : REAL := 0.0;
    robot6axis_ctrled1/robot6axis/armExtrem AT 22 : ARRAY[1..3] OF REAL := [3(0.0)];
    robot6axis_ctrled1/robot6axis/velX AT 21 : REAL := 0.0;
    robot6axis_ctrled1/robot6axis/velY AT 20 : REAL := 0.0;
    robot6axis_ctrled1/robot6axis/velZ AT 19 : REAL := 0.0;
    robot6axis_ctrled1/robot6axis/armInStop AT 5 : BOOL := false;
    robot6axis_ctrled1/robot6axis/servo_1/status AT 665 : INT := 0;
    robot6axis_ctrled1/robot6axis/servo_1/errorFlag AT 664 : INT := 0;
    robot6axis_ctrled1/robot6axis/servo_1/ActualPositionAx1 AT 6527 : REAL := 0.0;
    robot6axis_ctrled1/robot6axis/servo_1/MoveVelDone1 AT 234 : BOOL := false;
    robot6axis_ctrled1/robot6axis/servo_1/ActualVelocity1 AT 6526 : REAL := 0.0;
    robot6axis_ctrled1/robot6axis/servo_1/MoveAbsDone1 AT 233 : BOOL := false;
    robot6axis_ctrled1/robot6axis/servo_1/HomeCmd AT 98 : BOOL := false;
    robot6axis_ctrled1/robot6axis/servo_1/MoveVelCmd AT 97 : BOOL := false;
    robot6axis_ctrled1/robot6axis/servo_1/MoveAbsCmd AT 96 : BOOL := false;
    robot6axis_ctrled1/robot6axis/servo_1/MoveVel1ManualCmd AT 95 : BOOL := false;
    robot6axis_ctrled1/robot6axis/servo_1/MoveVel2ManualCmd AT 94 : BOOL := false;
    robot6axis_ctrled1/robot6axis/servo_1/MoveAbs1ManualCmd AT 93 : BOOL := false;
    robot6axis_ctrled1/robot6axis/servo_1/MoveAbs2ManualCmd AT 92 : BOOL := false;
    robot6axis_ctrled1/robot6axis/servo_1/StopCmd AT 22 : BOOL := false;
    robot6axis_ctrled1/robot6axis/servo_1/MovePosition AT 93 : REAL := 0.0;
    robot6axis_ctrled1/robot6axis/servo_1/MoveSpeed AT 92 : REAL := 100.0;
    robot6axis_ctrled1/robot6axis/servo_1/MoveAcceleration AT 91 : REAL := 100.0;
    robot6axis_ctrled1/robot6axis/servo_1/MoveDeceleration AT 90 : REAL := 100.0;
    robot6axis_ctrled1/robot6axis/servo_1/offsetAxToMa AT 89 : REAL := 0.0;
    robot6axis_ctrled1/robot6axis/servo_1/PLC_StatusReady AT 56 : BOOL := true;
    robot6axis_ctrled1/robot6axis/servo_1/PLC_StatusMoved AT 55 : BOOL := false;
    robot6axis_ctrled1/robot6axis/servo_1/PLC_StatusStand AT 54 : BOOL := false;
    robot6axis_ctrled1/robot6axis/servo_1/PLC_ActualPositionAx AT 167 : REAL := 0.0;
    robot6axis_ctrled1/robot6axis/servo_1/PLC_ActualPositionMa AT 63 : REAL := 0.0;
    robot6axis_ctrled1/robot6axis/servo_1/PLC_ActualVelocity AT 62 : REAL := 0.0;
    robot6axis_ctrled1/robot6axis/servo_1/physicalPosInit AT 6525 : REAL := 0.0;
    robot6axis_ctrled1/robot6axis/servo_1/MAX_SPEED AT 6524 : REAL(0.0..3.4e+038) := 30.0;
    robot6axis_ctrled1/robot6axis/servo_1/MAX_ACCEL AT 6523 : REAL(0.0..3.4e+038) := 1500.0;
    robot6axis_ctrled1/robot6axis/servo_1/MAX_DECEL AT 6522 : REAL(0.0..3.4e+038) := 1500.0;
    robot6axis_ctrled1/robot6axis/servo_1/MODULO_LENGTH AT 6521 : REAL := 0.0;
    robot6axis_ctrled1/robot6axis/servo_1/StatusReady AT 232 : BOOL := true;
    robot6axis_ctrled1/robot6axis/servo_1/StatusMoved AT 231 : BOOL := false;
    robot6axis_ctrled1/robot6axis/servo_1/StatusStand AT 230 : BOOL := false;
    robot6axis_ctrled1/robot6axis/servo_1/ActualPositionAx AT 6528 : REAL := 0.0;
    robot6axis_ctrled1/robot6axis/servo_1/ActualPositionMa AT 6520 : REAL := 0.0;
    robot6axis_ctrled1/robot6axis/servo_1/ActualVelocity AT 51 : REAL := 0.0;
    robot6axis_ctrled1/robot6axis/servo_1/MaximumVelocity AT 6519 : REAL := 0.0;
    robot6axis_ctrled1/robot6axis/servo_1/StatusPosIncrease AT 229 : BOOL := false;
    robot6axis_ctrled1/robot6axis/servo_1/StatusPosDecrease AT 228 : BOOL := false;
    robot6axis_ctrled1/robot6axis/servo_1/displayJauge AT 6518 : REAL := 0.0;
    robot6axis_ctrled1/robot6axis/servo_1/servo_mode/PLC_StatusReady AT 56 : BOOL := true;
    robot6axis_ctrled1/robot6axis/servo_1/servo_mode/PLC_StatusMoved AT 55 : BOOL := false;
    robot6axis_ctrled1/robot6axis/servo_1/servo_mode/PLC_StatusStand AT 54 : BOOL := false;
    robot6axis_ctrled1/robot6axis/servo_1/servo_mode/PLC_ActualPositionAx AT 167 : REAL := 0.0;
    robot6axis_ctrled1/robot6axis/servo_1/servo_mode/PLC_ActualPositionMa AT 63 : REAL := 0.0;
    robot6axis_ctrled1/robot6axis/servo_1/servo_mode/PLC_ActualVelocity AT 62 : REAL := 0.0;
    robot6axis_ctrled1/robot6axis/servo_1/servo_mode/StatusReady AT 235 : BOOL := true;
    robot6axis_ctrled1/robot6axis/servo_1/servo_mode/StatusMoved AT 236 : BOOL := false;
    robot6axis_ctrled1/robot6axis/servo_1/servo_mode/StatusStand AT 237 : BOOL := false;
    robot6axis_ctrled1/robot6axis/servo_1/servo_mode/ActualPositionMa AT 6617 : REAL := 0.0;
    robot6axis_ctrled1/robot6axis/servo_1/servo_mode/ActualVelocity AT 6618 : REAL := 0.0;
    robot6axis_ctrled1/robot6axis/servo_1/servo_mode/MaximumVelocity AT 6619 : REAL := 0.0;
    robot6axis_ctrled1/robot6axis/servo_1/servo_mode/physicalPosInit AT 6525 : REAL := 0.0;
    robot6axis_ctrled1/robot6axis/servo_1/servo_mode/ActualPositionAx AT 6527 : REAL := 0.0;
    robot6axis_ctrled1/robot6axis/servo_1/servo_mode/StatusReady_o AT 232 : BOOL := true;
    robot6axis_ctrled1/robot6axis/servo_1/servo_mode/StatusMoved_o AT 231 : BOOL := false;
    robot6axis_ctrled1/robot6axis/servo_1/servo_mode/StatusStand_o AT 230 : BOOL := false;
    robot6axis_ctrled1/robot6axis/servo_1/servo_mode/ActualPositionAx_o AT 6528 : REAL := 0.0;
    robot6axis_ctrled1/robot6axis/servo_1/servo_mode/ActualPositionMa_o AT 6520 : REAL := 0.0;
    robot6axis_ctrled1/robot6axis/servo_1/servo_mode/ActualVelocity_o AT 51 : REAL := 0.0;
    robot6axis_ctrled1/robot6axis/servo_1/servo_mode/MaximumVelocity_o AT 6519 : REAL := 0.0;
    robot6axis_ctrled1/robot6axis/servo_1/servo_mode/StatusPosIncrease_o AT 229 : BOOL := false;
    robot6axis_ctrled1/robot6axis/servo_1/servo_mode/StatusPosDecrease_o AT 228 : BOOL := false;
    robot6axis_ctrled1/robot6axis/servo_1/servo_mode/displayJauge_o AT 6518 : REAL := 0.0;
    robot6axis_ctrled1/robot6axis/servo_1/servo_mode/PLCMode AT 242 : BOOL := false;
    robot6axis_ctrled1/robot6axis/servo_1/servo_mode/PLCMode1 AT 243 : BOOL := false;
    robot6axis_ctrled1/robot6axis/servo_1/servo_mode/initDone AT 244 : BOOL := false;
    robot6axis_ctrled1/robot6axis/servo_1/servo_mode/displayPosMin AT 6622 : REAL := 0.0;
    robot6axis_ctrled1/robot6axis/servo_1/servo_mode/displayPosMax AT 6623 : REAL := 0.0;
    robot6axis_ctrled1/robot6axis/servo_1/servo_mode/PLC_ActualPositionAx1 AT 6624 : REAL := 0.0;
    robot6axis_ctrled1/robot6axis/servo_1/servo_mode/PLC_ActualVelocity1 AT 6625 : REAL := 0.0;
    robot6axis_ctrled1/robot6axis/servo_1/servo_mode/ActualPositionAx1 AT 6626 : REAL := 0.0;
    robot6axis_ctrled1/robot6axis/servo_1/servo_mode/ActualVelocity1 AT 6627 : REAL := 0.0;
    robot6axis_ctrled1/robot6axis/servo_1/servo_mode/offsetAxToMa AT 6628 : REAL := 0.0;
    robot6axis_ctrled1/robot6axis/servo_1/servo_mode/offsetAxToMa1 AT 6629 : REAL := 0.0;
    robot6axis_ctrled1/robot6axis/servo_1/servo_mode/ActualPositionMa_o1 AT 6630 : REAL := 0.0;
    robot6axis_ctrled1/robot6axis/servo_1/servo_control/HomeCmd AT 98 : BOOL := false;
    robot6axis_ctrled1/robot6axis/servo_1/servo_control/MoveVelCmd AT 97 : BOOL := false;
    robot6axis_ctrled1/robot6axis/servo_1/servo_control/MoveAbsCmd AT 96 : BOOL := false;
    robot6axis_ctrled1/robot6axis/servo_1/servo_control/MoveVel1ManualCmd AT 95 : BOOL := false;
    robot6axis_ctrled1/robot6axis/servo_1/servo_control/MoveVel2ManualCmd AT 94 : BOOL := false;
    robot6axis_ctrled1/robot6axis/servo_1/servo_control/MoveAbs1ManualCmd AT 93 : BOOL := false;
    robot6axis_ctrled1/robot6axis/servo_1/servo_control/MoveAbs2ManualCmd AT 92 : BOOL := false;
    robot6axis_ctrled1/robot6axis/servo_1/servo_control/StopCmd AT 22 : BOOL := false;
    robot6axis_ctrled1/robot6axis/servo_1/servo_control/MovePosition AT 93 : REAL := 0.0;
    robot6axis_ctrled1/robot6axis/servo_1/servo_control/MoveSpeed AT 92 : REAL := 100.0;
    robot6axis_ctrled1/robot6axis/servo_1/servo_control/MoveAcceleration AT 91 : REAL := 100.0;
    robot6axis_ctrled1/robot6axis/servo_1/servo_control/MoveDeceleration AT 90 : REAL := 100.0;
    robot6axis_ctrled1/robot6axis/servo_1/servo_control/offsetAxToMa AT 89 : REAL := 0.0;
    robot6axis_ctrled1/robot6axis/servo_1/servo_control/physicalPosInit AT 6525 : REAL := 0.0;
    robot6axis_ctrled1/robot6axis/servo_1/servo_control/MAX_SPEED AT 6524 : REAL(0.0..3.4e+038) := 30.0;
    robot6axis_ctrled1/robot6axis/servo_1/servo_control/status AT 665 : INT := 0;
    robot6axis_ctrled1/robot6axis/servo_1/servo_control/errorFlag AT 664 : INT := 0;
    robot6axis_ctrled1/robot6axis/servo_1/servo_control/IOActualPositionAx AT 6527 : REAL := 0.0;
    robot6axis_ctrled1/robot6axis/servo_1/servo_control/IOVelDone AT 234 : BOOL := false;
    robot6axis_ctrled1/robot6axis/servo_1/servo_control/IOAbsDone AT 233 : BOOL := false;
    robot6axis_ctrled1/robot6axis/servo_1/servo_control/IOActualVelocity AT 6526 : REAL := 0.0;
    robot6axis_ctrled1/robot6axis/servo_1/servo_control/OperationMode AT 667 : INT := 0;
    robot6axis_ctrled1/robot6axis/servo_1/servo_control/StatusReady AT 235 : BOOL := true;
    robot6axis_ctrled1/robot6axis/servo_1/servo_control/StatusMove AT 236 : BOOL := false;
    robot6axis_ctrled1/robot6axis/servo_1/servo_control/StatusStand AT 237 : BOOL := false;
    robot6axis_ctrled1/robot6axis/servo_1/servo_control/ActualPositionMa AT 6617 : REAL := 0.0;
    robot6axis_ctrled1/robot6axis/servo_1/servo_control/ActualVelocity AT 6618 : REAL := 0.0;
    robot6axis_ctrled1/robot6axis/servo_1/servo_control/MaximumVelocity AT 6619 : REAL := 0.0;
    robot6axis_ctrled1/robot6axis/servo_1/servo_control/VelEnabled AT 238 : BOOL := false;
    robot6axis_ctrled1/robot6axis/servo_1/servo_control/VelCmd AT 239 : BOOL := false;
    robot6axis_ctrled1/robot6axis/servo_1/servo_control/PosEnabled AT 240 : BOOL := false;
    robot6axis_ctrled1/robot6axis/servo_1/servo_control/PosCmd AT 241 : BOOL := false;
    robot6axis_ctrled1/robot6axis/servo_1/servo_control/Position AT 6621 : REAL := 0.0;
    robot6axis_ctrled1/robot6axis/servo_1/servo_control/Speed AT 6620 : REAL := 0.0;
    robot6axis_ctrled1/robot6axis/servo_1/servo_control/ManualMode AT 668 : INT := 0;
    robot6axis_ctrled1/robot6axis/servo_1/servo_control/initDone AT 245 : BOOL := false;
    robot6axis_ctrled1/robot6axis/servo_1/servo_control/ActualPositionMa1 AT 6631 : REAL := 0.0;
    robot6axis_ctrled1/robot6axis/servo_1/servo_control/offsetAxToMa1 AT 6632 : REAL := 0.0;
    robot6axis_ctrled1/robot6axis/servo_1/servo_control/HOME_POSITION AT 6633 : REAL := 100.0;
    robot6axis_ctrled1/robot6axis/servo_1/servo_control/MANUAL_POSITION1 AT 6634 : REAL := 0.0;
    robot6axis_ctrled1/robot6axis/servo_1/servo_control/MANUAL_POSITION2 AT 6635 : REAL := 150.0;
    robot6axis_ctrled1/robot6axis/servo_1/servo_control/MANUAL_SPEED1 AT 6636 : REAL := -100.0;
    robot6axis_ctrled1/robot6axis/servo_1/servo_control/MANUAL_SPEED2 AT 6637 : REAL := 100.0;
    robot6axis_ctrled1/robot6axis/servo_1/servo_control/MANUAL_SPEED AT 6638 : REAL := 100.0;
    robot6axis_ctrled1/robot6axis/servo_1/servo_velocity/MoveVelEnable AT 238 : BOOL := false;
    robot6axis_ctrled1/robot6axis/servo_1/servo_velocity/MoveVelStart AT 239 : BOOL := false;
    robot6axis_ctrled1/robot6axis/servo_1/servo_velocity/MoveSpeed AT 6620 : REAL := 0.0;
    robot6axis_ctrled1/robot6axis/servo_1/servo_velocity/MoveAcceleration AT 91 : REAL := 100.0;
    robot6axis_ctrled1/robot6axis/servo_1/servo_velocity/MoveDeceleration AT 90 : REAL := 100.0;
    robot6axis_ctrled1/robot6axis/servo_1/servo_velocity/MAX_SPEED AT 6524 : REAL(0.0..3.4e+038) := 30.0;
    robot6axis_ctrled1/robot6axis/servo_1/servo_velocity/MAX_ACCEL AT 6523 : REAL(0.0..3.4e+038) := 1500.0;
    robot6axis_ctrled1/robot6axis/servo_1/servo_velocity/MAX_DECEL AT 6522 : REAL(0.0..3.4e+038) := 1500.0;
    robot6axis_ctrled1/robot6axis/servo_1/servo_velocity/MODULO_LENGTH AT 6521 : REAL := 0.0;
    robot6axis_ctrled1/robot6axis/servo_1/servo_velocity/status AT 665 : INT := 0;
    robot6axis_ctrled1/robot6axis/servo_1/servo_velocity/errorFlag AT 664 : INT := 0;
    robot6axis_ctrled1/robot6axis/servo_1/servo_velocity/MoveVelDone AT 234 : BOOL := false;
    robot6axis_ctrled1/robot6axis/servo_1/servo_velocity/ActualPositionAx AT 6527 : REAL := 0.0;
    robot6axis_ctrled1/robot6axis/servo_1/servo_velocity/ActualVelocity AT 6526 : REAL := 0.0;
    robot6axis_ctrled1/robot6axis/servo_1/servo_velocity/firstStep AT 246 : BOOL := true;
    robot6axis_ctrled1/robot6axis/servo_1/servo_velocity/stepDone AT 247 : BOOL := false;
    robot6axis_ctrled1/robot6axis/servo_1/servo_velocity/currentTime AT 6639 : REAL := 0.0;
    robot6axis_ctrled1/robot6axis/servo_1/servo_velocity/MoveSpeed1 AT 6640 : REAL := 0.0;
    robot6axis_ctrled1/robot6axis/servo_1/servo_velocity/acceleration AT 6641 : REAL := 0.0;
    robot6axis_ctrled1/robot6axis/servo_1/servo_velocity/deceleration AT 6642 : REAL := 0.0;
    robot6axis_ctrled1/robot6axis/servo_1/servo_velocity/orderSpeed AT 6643 : REAL := 0.0;
    robot6axis_ctrled1/robot6axis/servo_1/servo_velocity/endChangeSpeed AT 6644 : REAL := 0.0;
    robot6axis_ctrled1/robot6axis/servo_1/servo_velocity/accelDecelChangeSpeed AT 6645 : REAL := 0.0;
    robot6axis_ctrled1/robot6axis/servo_1/servo_velocity/ActualVelocity1 AT 6646 : REAL := 0.0;
    robot6axis_ctrled1/robot6axis/servo_1/servo_velocity/speedChanged AT 248 : BOOL := false;
    robot6axis_ctrled1/robot6axis/servo_1/servo_position/MoveAbsEnable AT 240 : BOOL := false;
    robot6axis_ctrled1/robot6axis/servo_1/servo_position/MoveAbsStart AT 241 : BOOL := false;
    robot6axis_ctrled1/robot6axis/servo_1/servo_position/MovePosition AT 6621 : REAL := 0.0;
    robot6axis_ctrled1/robot6axis/servo_1/servo_position/MoveSpeed AT 6620 : REAL := 0.0;
    robot6axis_ctrled1/robot6axis/servo_1/servo_position/MoveAcceleration AT 91 : REAL := 100.0;
    robot6axis_ctrled1/robot6axis/servo_1/servo_position/MoveDeceleration AT 90 : REAL := 100.0;
    robot6axis_ctrled1/robot6axis/servo_1/servo_position/MAX_SPEED AT 6524 : REAL(0.0..3.4e+038) := 30.0;
    robot6axis_ctrled1/robot6axis/servo_1/servo_position/MAX_ACCEL AT 6523 : REAL(0.0..3.4e+038) := 1500.0;
    robot6axis_ctrled1/robot6axis/servo_1/servo_position/MAX_DECEL AT 6522 : REAL(0.0..3.4e+038) := 1500.0;
    robot6axis_ctrled1/robot6axis/servo_1/servo_position/MODULO_LENGTH AT 6521 : REAL := 0.0;
    robot6axis_ctrled1/robot6axis/servo_1/servo_position/status AT 665 : INT := 0;
    robot6axis_ctrled1/robot6axis/servo_1/servo_position/errorFlag AT 664 : INT := 0;
    robot6axis_ctrled1/robot6axis/servo_1/servo_position/MoveAbsDone AT 233 : BOOL := false;
    robot6axis_ctrled1/robot6axis/servo_1/servo_position/ActualPositionAx AT 6527 : REAL := 0.0;
    robot6axis_ctrled1/robot6axis/servo_1/servo_position/ActualVelocity AT 6526 : REAL := 0.0;
    robot6axis_ctrled1/robot6axis/servo_1/servo_position/firstStep AT 249 : BOOL := true;
    robot6axis_ctrled1/robot6axis/servo_1/servo_position/stepDone AT 250 : BOOL := false;
    robot6axis_ctrled1/robot6axis/servo_1/servo_position/timeToStop AT 6647 : REAL := 0.0;
    robot6axis_ctrled1/robot6axis/servo_1/servo_position/distanceToStop AT 6648 : REAL := 0.0;
    robot6axis_ctrled1/robot6axis/servo_1/servo_position/distance AT 6649 : REAL := 0.0;
    robot6axis_ctrled1/robot6axis/servo_1/servo_position/currentTime AT 6650 : REAL := 0.0;
    robot6axis_ctrled1/robot6axis/servo_1/servo_position/currentSpeed1 AT 6651 : REAL := 0.0;
    robot6axis_ctrled1/robot6axis/servo_1/servo_position/targetPosition AT 6652 : REAL := 0.0;
    robot6axis_ctrled1/robot6axis/servo_1/servo_position/ActualPositionAx1 AT 6653 : REAL := 0.0;
    robot6axis_ctrled1/robot6axis/servo_1/servo_position/acceleration AT 6654 : REAL := 0.0;
    robot6axis_ctrled1/robot6axis/servo_1/servo_position/deceleration AT 6655 : REAL := 0.0;
    robot6axis_ctrled1/robot6axis/servo_1/servo_position/orderSpeed AT 6656 : REAL := 0.0;
    robot6axis_ctrled1/robot6axis/servo_1/servo_position/moveDirection AT 6657 : REAL := 0.0;
    robot6axis_ctrled1/robot6axis/servo_1/servo_position/moveDirection1 AT 6658 : REAL := 0.0;
    robot6axis_ctrled1/robot6axis/servo_1/servo_position/endChangeSpeed AT 6659 : REAL := 0.0;
    robot6axis_ctrled1/robot6axis/servo_1/servo_position/ActualVelocity1 AT 6660 : REAL := 0.0;
    robot6axis_ctrled1/robot6axis/FOOT/armOrigin AT 27 : ARRAY[1..3] OF REAL := [800.0, 400.0, 0.0];
    robot6axis_ctrled1/robot6axis/FOOT/overallArmQuatInput AT 6512 : ARRAY[1..4] OF REAL := [1.0, 3(0.0)];
    robot6axis_ctrled1/robot6axis/FOOT/structRotVector AT 162 : ARRAY[1..3] OF REAL := [0.0, 1.0, 0.0];
    robot6axis_ctrled1/robot6axis/FOOT/structRotDeg AT 161 : REAL := -90.01;
    robot6axis_ctrled1/robot6axis/FOOT/driveRotVector AT 143 : ARRAY[1..3] OF REAL := [1.0, 2(0.0)];
    robot6axis_ctrled1/robot6axis/FOOT/driveRotDeg AT 6528 : REAL := 0.0;
    robot6axis_ctrled1/robot6axis/FOOT/ownRotDeg AT 160 : REAL := 90.0;
    robot6axis_ctrled1/robot6axis/FOOT/driveResizeLength AT 6511 : REAL := 0.0;
    robot6axis_ctrled1/robot6axis/FOOT/functionActive AT 227 : BOOL := false;
    robot6axis_ctrled1/robot6axis/FOOT/armExtrem AT 6529 : ARRAY[1..3] OF REAL := [3(0.0)];
    robot6axis_ctrled1/robot6axis/FOOT/overallArmRotOutput AT 6534 : ARRAY[1..4] OF REAL := [4(0.0)];
    robot6axis_ctrled1/robot6axis/FOOT/productId AT 663 : DINT := -1;
    robot6axis_ctrled1/robot6axis/FOOT/status_act_prod AT 669 : DINT := 0;
    robot6axis_ctrled1/robot6axis/FOOT/m11 AT 6661 : REAL := 1.0;
    robot6axis_ctrled1/robot6axis/FOOT/m12 AT 6662 : REAL := 0.0;
    robot6axis_ctrled1/robot6axis/FOOT/m13 AT 6663 : REAL := 0.0;
    robot6axis_ctrled1/robot6axis/FOOT/m14 AT 6664 : REAL := 0.0;
    robot6axis_ctrled1/robot6axis/FOOT/m21 AT 6665 : REAL := 0.0;
    robot6axis_ctrled1/robot6axis/FOOT/m22 AT 6666 : REAL := 1.0;
    robot6axis_ctrled1/robot6axis/FOOT/m23 AT 6667 : REAL := 0.0;
    robot6axis_ctrled1/robot6axis/FOOT/m24 AT 6668 : REAL := 0.0;
    robot6axis_ctrled1/robot6axis/FOOT/m31 AT 6669 : REAL := 0.0;
    robot6axis_ctrled1/robot6axis/FOOT/m32 AT 6670 : REAL := 0.0;
    robot6axis_ctrled1/robot6axis/FOOT/m33 AT 6671 : REAL := 1.0;
    robot6axis_ctrled1/robot6axis/FOOT/m34 AT 6672 : REAL := 0.0;
    robot6axis_ctrled1/robot6axis/FOOT/m41 AT 6673 : REAL := 0.0;
    robot6axis_ctrled1/robot6axis/FOOT/m42 AT 6674 : REAL := 0.0;
    robot6axis_ctrled1/robot6axis/FOOT/m43 AT 6675 : REAL := 0.0;
    robot6axis_ctrled1/robot6axis/FOOT/m44 AT 6676 : REAL := 1.0;
    robot6axis_ctrled1/robot6axis/FOOT/armLengthCalc AT 6677 : REAL := 0.0;
    robot6axis_ctrled1/robot6axis/FOOT/functionActiveLocale AT 251 : BOOL := false;
    robot6axis_ctrled1/robot6axis/FOOT/product_id AT 670 : DINT := -1;
    robot6axis_ctrled1/robot6axis/FOOT/arm_id AT 671 : DINT := -1;
    robot6axis_ctrled1/robot6axis/FOOT/timeToGripParam AT 6678 : REAL := 0.15;
    robot6axis_ctrled1/robot6axis/FOOT/armLength AT 6679 : REAL := 375.0;
    robot6axis_ctrled1/robot6axis/FOOT/armWidth AT 6680 : REAL := 60.0;
    robot6axis_ctrled1/robot6axis/FOOT/armHeight AT 6681 : REAL := 60.0;
    robot6axis_ctrled1/robot6axis/FOOT/armType AT 672 : INT := 0;
    robot6axis_ctrled1/robot6axis/FOOT2/armOrigin AT 6529 : ARRAY[1..3] OF REAL := [3(0.0)];
    robot6axis_ctrled1/robot6axis/FOOT2/overallArmQuatInput AT 6534 : ARRAY[1..4] OF REAL := [4(0.0)];
    robot6axis_ctrled1/robot6axis/FOOT2/structRotVector AT 155 : ARRAY[1..3] OF REAL := [2(0.0), 1.0];
    robot6axis_ctrled1/robot6axis/FOOT2/structRotDeg AT 154 : REAL := 90.0;
    robot6axis_ctrled1/robot6axis/FOOT2/driveRotVector AT 6506 : ARRAY[1..3] OF REAL := [2(0.0), 1.0];
    robot6axis_ctrled1/robot6axis/FOOT2/driveRotDeg AT 6505 : REAL := 0.0;
    robot6axis_ctrled1/robot6axis/FOOT2/ownRotDeg AT 6504 : REAL := 0.0;
    robot6axis_ctrled1/robot6axis/FOOT2/driveResizeLength AT 6503 : REAL := 0.0;
    robot6axis_ctrled1/robot6axis/FOOT2/functionActive AT 226 : BOOL := false;
    robot6axis_ctrled1/robot6axis/FOOT2/armExtrem AT 6540 : ARRAY[1..3] OF REAL := [3(0.0)];
    robot6axis_ctrled1/robot6axis/FOOT2/overallArmRotOutput AT 6545 : ARRAY[1..4] OF REAL := [4(0.0)];
    robot6axis_ctrled1/robot6axis/FOOT2/productId AT 662 : DINT := -1;
    robot6axis_ctrled1/robot6axis/FOOT2/status_act_prod AT 673 : DINT := 0;
    robot6axis_ctrled1/robot6axis/FOOT2/m11 AT 6682 : REAL := 1.0;
    robot6axis_ctrled1/robot6axis/FOOT2/m12 AT 6683 : REAL := 0.0;
    robot6axis_ctrled1/robot6axis/FOOT2/m13 AT 6684 : REAL := 0.0;
    robot6axis_ctrled1/robot6axis/FOOT2/m14 AT 6685 : REAL := 0.0;
    robot6axis_ctrled1/robot6axis/FOOT2/m21 AT 6686 : REAL := 0.0;
    robot6axis_ctrled1/robot6axis/FOOT2/m22 AT 6687 : REAL := 1.0;
    robot6axis_ctrled1/robot6axis/FOOT2/m23 AT 6688 : REAL := 0.0;
    robot6axis_ctrled1/robot6axis/FOOT2/m24 AT 6689 : REAL := 0.0;
    robot6axis_ctrled1/robot6axis/FOOT2/m31 AT 6690 : REAL := 0.0;
    robot6axis_ctrled1/robot6axis/FOOT2/m32 AT 6691 : REAL := 0.0;
    robot6axis_ctrled1/robot6axis/FOOT2/m33 AT 6692 : REAL := 1.0;
    robot6axis_ctrled1/robot6axis/FOOT2/m34 AT 6693 : REAL := 0.0;
    robot6axis_ctrled1/robot6axis/FOOT2/m41 AT 6694 : REAL := 0.0;
    robot6axis_ctrled1/robot6axis/FOOT2/m42 AT 6695 : REAL := 0.0;
    robot6axis_ctrled1/robot6axis/FOOT2/m43 AT 6696 : REAL := 0.0;
    robot6axis_ctrled1/robot6axis/FOOT2/m44 AT 6697 : REAL := 1.0;
    robot6axis_ctrled1/robot6axis/FOOT2/armLengthCalc AT 6698 : REAL := 0.0;
    robot6axis_ctrled1/robot6axis/FOOT2/functionActiveLocale AT 252 : BOOL := false;
    robot6axis_ctrled1/robot6axis/FOOT2/product_id AT 674 : DINT := -1;
    robot6axis_ctrled1/robot6axis/FOOT2/arm_id AT 675 : DINT := -1;
    robot6axis_ctrled1/robot6axis/FOOT2/timeToGripParam AT 6699 : REAL := 0.15;
    robot6axis_ctrled1/robot6axis/FOOT2/armLength AT 6700 : REAL := 20.0;
    robot6axis_ctrled1/robot6axis/FOOT2/armWidth AT 6701 : REAL := 60.0;
    robot6axis_ctrled1/robot6axis/FOOT2/armHeight AT 6702 : REAL := 60.0;
    robot6axis_ctrled1/robot6axis/FOOT2/armType AT 676 : INT := 0;
    robot6axis_ctrled1/robot6axis/servo_2/status AT 661 : INT := 0;
    robot6axis_ctrled1/robot6axis/servo_2/errorFlag AT 660 : INT := 0;
    robot6axis_ctrled1/robot6axis/servo_2/ActualPositionAx1 AT 6502 : REAL := 0.0;
    robot6axis_ctrled1/robot6axis/servo_2/MoveVelDone1 AT 225 : BOOL := false;
    robot6axis_ctrled1/robot6axis/servo_2/ActualVelocity1 AT 6501 : REAL := 0.0;
    robot6axis_ctrled1/robot6axis/servo_2/MoveAbsDone1 AT 224 : BOOL := false;
    robot6axis_ctrled1/robot6axis/servo_2/HomeCmd AT 91 : BOOL := false;
    robot6axis_ctrled1/robot6axis/servo_2/MoveVelCmd AT 90 : BOOL := false;
    robot6axis_ctrled1/robot6axis/servo_2/MoveAbsCmd AT 89 : BOOL := false;
    robot6axis_ctrled1/robot6axis/servo_2/MoveVel1ManualCmd AT 88 : BOOL := false;
    robot6axis_ctrled1/robot6axis/servo_2/MoveVel2ManualCmd AT 87 : BOOL := false;
    robot6axis_ctrled1/robot6axis/servo_2/MoveAbs1ManualCmd AT 86 : BOOL := false;
    robot6axis_ctrled1/robot6axis/servo_2/MoveAbs2ManualCmd AT 85 : BOOL := false;
    robot6axis_ctrled1/robot6axis/servo_2/StopCmd AT 22 : BOOL := false;
    robot6axis_ctrled1/robot6axis/servo_2/MovePosition AT 88 : REAL := 0.0;
    robot6axis_ctrled1/robot6axis/servo_2/MoveSpeed AT 87 : REAL := 100.0;
    robot6axis_ctrled1/robot6axis/servo_2/MoveAcceleration AT 86 : REAL := 100.0;
    robot6axis_ctrled1/robot6axis/servo_2/MoveDeceleration AT 85 : REAL := 100.0;
    robot6axis_ctrled1/robot6axis/servo_2/offsetAxToMa AT 84 : REAL := 0.0;
    robot6axis_ctrled1/robot6axis/servo_2/PLC_StatusReady AT 53 : BOOL := true;
    robot6axis_ctrled1/robot6axis/servo_2/PLC_StatusMoved AT 52 : BOOL := false;
    robot6axis_ctrled1/robot6axis/servo_2/PLC_StatusStand AT 51 : BOOL := false;
    robot6axis_ctrled1/robot6axis/servo_2/PLC_ActualPositionAx AT 168 : REAL := 0.0;
    robot6axis_ctrled1/robot6axis/servo_2/PLC_ActualPositionMa AT 61 : REAL := 0.0;
    robot6axis_ctrled1/robot6axis/servo_2/PLC_ActualVelocity AT 60 : REAL := 0.0;
    robot6axis_ctrled1/robot6axis/servo_2/physicalPosInit AT 6500 : REAL := 0.0;
    robot6axis_ctrled1/robot6axis/servo_2/MAX_SPEED AT 6499 : REAL(0.0..3.4e+038) := 30.0;
    robot6axis_ctrled1/robot6axis/servo_2/MAX_ACCEL AT 6498 : REAL(0.0..3.4e+038) := 1500.0;
    robot6axis_ctrled1/robot6axis/servo_2/MAX_DECEL AT 6497 : REAL(0.0..3.4e+038) := 1500.0;
    robot6axis_ctrled1/robot6axis/servo_2/MODULO_LENGTH AT 6496 : REAL := 0.0;
    robot6axis_ctrled1/robot6axis/servo_2/StatusReady AT 223 : BOOL := true;
    robot6axis_ctrled1/robot6axis/servo_2/StatusMoved AT 222 : BOOL := false;
    robot6axis_ctrled1/robot6axis/servo_2/StatusStand AT 221 : BOOL := false;
    robot6axis_ctrled1/robot6axis/servo_2/ActualPositionAx AT 6551 : REAL := 0.0;
    robot6axis_ctrled1/robot6axis/servo_2/ActualPositionMa AT 6495 : REAL := 0.0;
    robot6axis_ctrled1/robot6axis/servo_2/ActualVelocity AT 50 : REAL := 0.0;
    robot6axis_ctrled1/robot6axis/servo_2/MaximumVelocity AT 6494 : REAL := 0.0;
    robot6axis_ctrled1/robot6axis/servo_2/StatusPosIncrease AT 220 : BOOL := false;
    robot6axis_ctrled1/robot6axis/servo_2/StatusPosDecrease AT 219 : BOOL := false;
    robot6axis_ctrled1/robot6axis/servo_2/displayJauge AT 6493 : REAL := 0.0;
    robot6axis_ctrled1/robot6axis/servo_2/servo_mode/PLC_StatusReady AT 53 : BOOL := true;
    robot6axis_ctrled1/robot6axis/servo_2/servo_mode/PLC_StatusMoved AT 52 : BOOL := false;
    robot6axis_ctrled1/robot6axis/servo_2/servo_mode/PLC_StatusStand AT 51 : BOOL := false;
    robot6axis_ctrled1/robot6axis/servo_2/servo_mode/PLC_ActualPositionAx AT 168 : REAL := 0.0;
    robot6axis_ctrled1/robot6axis/servo_2/servo_mode/PLC_ActualPositionMa AT 61 : REAL := 0.0;
    robot6axis_ctrled1/robot6axis/servo_2/servo_mode/PLC_ActualVelocity AT 60 : REAL := 0.0;
    robot6axis_ctrled1/robot6axis/servo_2/servo_mode/StatusReady AT 253 : BOOL := true;
    robot6axis_ctrled1/robot6axis/servo_2/servo_mode/StatusMoved AT 254 : BOOL := false;
    robot6axis_ctrled1/robot6axis/servo_2/servo_mode/StatusStand AT 255 : BOOL := false;
    robot6axis_ctrled1/robot6axis/servo_2/servo_mode/ActualPositionMa AT 6703 : REAL := 0.0;
    robot6axis_ctrled1/robot6axis/servo_2/servo_mode/ActualVelocity AT 6704 : REAL := 0.0;
    robot6axis_ctrled1/robot6axis/servo_2/servo_mode/MaximumVelocity AT 6705 : REAL := 0.0;
    robot6axis_ctrled1/robot6axis/servo_2/servo_mode/physicalPosInit AT 6500 : REAL := 0.0;
    robot6axis_ctrled1/robot6axis/servo_2/servo_mode/ActualPositionAx AT 6502 : REAL := 0.0;
    robot6axis_ctrled1/robot6axis/servo_2/servo_mode/StatusReady_o AT 223 : BOOL := true;
    robot6axis_ctrled1/robot6axis/servo_2/servo_mode/StatusMoved_o AT 222 : BOOL := false;
    robot6axis_ctrled1/robot6axis/servo_2/servo_mode/StatusStand_o AT 221 : BOOL := false;
    robot6axis_ctrled1/robot6axis/servo_2/servo_mode/ActualPositionAx_o AT 6551 : REAL := 0.0;
    robot6axis_ctrled1/robot6axis/servo_2/servo_mode/ActualPositionMa_o AT 6495 : REAL := 0.0;
    robot6axis_ctrled1/robot6axis/servo_2/servo_mode/ActualVelocity_o AT 50 : REAL := 0.0;
    robot6axis_ctrled1/robot6axis/servo_2/servo_mode/MaximumVelocity_o AT 6494 : REAL := 0.0;
    robot6axis_ctrled1/robot6axis/servo_2/servo_mode/StatusPosIncrease_o AT 220 : BOOL := false;
    robot6axis_ctrled1/robot6axis/servo_2/servo_mode/StatusPosDecrease_o AT 219 : BOOL := false;
    robot6axis_ctrled1/robot6axis/servo_2/servo_mode/displayJauge_o AT 6493 : REAL := 0.0;
    robot6axis_ctrled1/robot6axis/servo_2/servo_mode/PLCMode AT 260 : BOOL := false;
    robot6axis_ctrled1/robot6axis/servo_2/servo_mode/PLCMode1 AT 261 : BOOL := false;
    robot6axis_ctrled1/robot6axis/servo_2/servo_mode/initDone AT 262 : BOOL := false;
    robot6axis_ctrled1/robot6axis/servo_2/servo_mode/displayPosMin AT 6708 : REAL := 0.0;
    robot6axis_ctrled1/robot6axis/servo_2/servo_mode/displayPosMax AT 6709 : REAL := 0.0;
    robot6axis_ctrled1/robot6axis/servo_2/servo_mode/PLC_ActualPositionAx1 AT 6710 : REAL := 0.0;
    robot6axis_ctrled1/robot6axis/servo_2/servo_mode/PLC_ActualVelocity1 AT 6711 : REAL := 0.0;
    robot6axis_ctrled1/robot6axis/servo_2/servo_mode/ActualPositionAx1 AT 6712 : REAL := 0.0;
    robot6axis_ctrled1/robot6axis/servo_2/servo_mode/ActualVelocity1 AT 6713 : REAL := 0.0;
    robot6axis_ctrled1/robot6axis/servo_2/servo_mode/offsetAxToMa AT 6714 : REAL := 0.0;
    robot6axis_ctrled1/robot6axis/servo_2/servo_mode/offsetAxToMa1 AT 6715 : REAL := 0.0;
    robot6axis_ctrled1/robot6axis/servo_2/servo_mode/ActualPositionMa_o1 AT 6716 : REAL := 0.0;
    robot6axis_ctrled1/robot6axis/servo_2/servo_control/HomeCmd AT 91 : BOOL := false;
    robot6axis_ctrled1/robot6axis/servo_2/servo_control/MoveVelCmd AT 90 : BOOL := false;
    robot6axis_ctrled1/robot6axis/servo_2/servo_control/MoveAbsCmd AT 89 : BOOL := false;
    robot6axis_ctrled1/robot6axis/servo_2/servo_control/MoveVel1ManualCmd AT 88 : BOOL := false;
    robot6axis_ctrled1/robot6axis/servo_2/servo_control/MoveVel2ManualCmd AT 87 : BOOL := false;
    robot6axis_ctrled1/robot6axis/servo_2/servo_control/MoveAbs1ManualCmd AT 86 : BOOL := false;
    robot6axis_ctrled1/robot6axis/servo_2/servo_control/MoveAbs2ManualCmd AT 85 : BOOL := false;
    robot6axis_ctrled1/robot6axis/servo_2/servo_control/StopCmd AT 22 : BOOL := false;
    robot6axis_ctrled1/robot6axis/servo_2/servo_control/MovePosition AT 88 : REAL := 0.0;
    robot6axis_ctrled1/robot6axis/servo_2/servo_control/MoveSpeed AT 87 : REAL := 100.0;
    robot6axis_ctrled1/robot6axis/servo_2/servo_control/MoveAcceleration AT 86 : REAL := 100.0;
    robot6axis_ctrled1/robot6axis/servo_2/servo_control/MoveDeceleration AT 85 : REAL := 100.0;
    robot6axis_ctrled1/robot6axis/servo_2/servo_control/offsetAxToMa AT 84 : REAL := 0.0;
    robot6axis_ctrled1/robot6axis/servo_2/servo_control/physicalPosInit AT 6500 : REAL := 0.0;
    robot6axis_ctrled1/robot6axis/servo_2/servo_control/MAX_SPEED AT 6499 : REAL(0.0..3.4e+038) := 30.0;
    robot6axis_ctrled1/robot6axis/servo_2/servo_control/status AT 661 : INT := 0;
    robot6axis_ctrled1/robot6axis/servo_2/servo_control/errorFlag AT 660 : INT := 0;
    robot6axis_ctrled1/robot6axis/servo_2/servo_control/IOActualPositionAx AT 6502 : REAL := 0.0;
    robot6axis_ctrled1/robot6axis/servo_2/servo_control/IOVelDone AT 225 : BOOL := false;
    robot6axis_ctrled1/robot6axis/servo_2/servo_control/IOAbsDone AT 224 : BOOL := false;
    robot6axis_ctrled1/robot6axis/servo_2/servo_control/IOActualVelocity AT 6501 : REAL := 0.0;
